(* PLC project CoDeSys External Library Template, WAGO e!COCKPIT e!COCKPIT, author 3S - Smart Software Solutions GmbH *)
(* stored: creationDateTime 2019-10-29T12:37:19.6730838, version 3.5.5.30, modificationDateTime 2019-10-29T12:36:39.3744516, organization 3S - Smart Software Solutions GmbH *)
(* Library project template with all possible element types, docu and a sample project structure *)

FUNCTION_BLOCK fbPPPSFriskoATTOM1S
  VAR_INPUT
    sKomunikat : alSTRINGKomunikat;  (* komunikat z systemu zewnętrznego *)
    intTablicaKomunikatowRozmiar : INT;  (* rozmiar tablicy danych wysyłkowych *)
    intModbusOdczytZapisZadanieRozmiar : INT;  (* rozmiar tablicy danych modbusa *)
    xTablicaKomunikatowHold : BOOL;  (* wstrzymanie komunikacji mniej ważnych komunikatów *)
    sIdInstancji : STRING;  (* parametr ID rolety np NS02L*202IBM**** *)
    sIdAplikacji : STRING;  (* parametr ID aplikacji np SO*******ECL*000 *)
    sMnemonik : STRING;  (* mnemonik właściciela - BCB* *)
    sMACAdres : STRING;  (* MAC adres sterownika *)
    sDaneZapasowe : STRING;  (* 6 znaków zapasu *)
    tCzasOpoznieniaRestartu : TIME;  (* czas opóźnienia po którym zaczynają być raportowane wartości *)
    tCzasOpoznieniaAlarmu : TIME := TIME#1m0s0ms;  (* czas opóźnienia po którym zaczynają być raportowane wartości *)
    bAdres : BYTE;
    tMinimalnyCzasRaportowania : TIME;
    tMaksymalnyCzasRaportowania : TIME;
    xAutonomizacja : BOOL;
    xAutonomizacjaSztuczna : BOOL;
    xSezonGrzewczyCalyRok : BOOL;
    rTemperaturaZasilaniaZadanaObieguCOKomfortAutonomizacja : REAL;  (* Domyślna wartość nastawy temperatury obiegu c.o. w trybie komfortowym *)
    rTemperaturaZasilaniaZadanaObieguCOEkonomicznaAutonomizacja : REAL;  (* Domyślna wartość nastawy temperatury obiegu c.o. w trybie ekonomicznym *)
  END_VAR
  VAR_IN_OUT
    arModbusOdczytCykliczny : ARRAY[1..5000] OF typModbusOdczytCykliczny;
    arModbusStatusKomunikacji : ARRAY[1..256] OF INT;
    arModbusOdczytZapisZadanie : ARRAY[1..1000] OF typModbusOdczytZapisZadanie;
    intModbusOdczytZapisZadanieZnacznikZapisu : INT;
    arTablicaKomunikatow : alARRAYTablicaKomunikatow;
    intTablicaKomunikatowZnacznikZapisu : INT;
    aTemperatury : ARRAY[0..96] OF REAL;  (* Tablica pomiarów temperatur bieżącego dnia *)
    rTemperaturaSrednia1Dzien : REAL;  (* Średnia dzienna temperatura *)
    iTemperaturyIndex : INT;  (* Index tablicy *)
    aTemperaturySrednie : ARRAY[0..2] OF REAL;  (* Tablica zawierająca średnie temperatury z trzech ostatnich dni *)
    iTemperaturySrednieIndex : INT;  (* Index tablicy śrenich temperatur *)
    rTemperaturaSrednia3Dni : REAL;  (* Średnia temperatura z trzech dni *)
    xTemperaturaSrednia3DniObliczona : BOOL;  (* Prawda, jeśli obliczona została średnia temperatura z trzech dni *)
  END_VAR
  VAR
    xPoInicjalizacji : BOOL := FALSE;  (* Inicjalizacja *)
    fbInicjalizacyjnyTimer : TON;
    tCzasInicjalizacji : TIME := TIME#30s0ms;
    xPierwszySkan : BOOL := TRUE;  (* Definicje zmiennych do odczytu wartości z modbusa *)
    intPetlaPierwszySkan : INT := 1;
    sDane : alSTRINGKomunikat;  (* Definicje do komunikacji z IZE *)
    sWyslanyKomunikat : alSTRINGKomunikat;
    sWyslanyKomunikatDummy : alSTRINGKomunikat;
    xZadanieRaportu : BOOL;
    sKomunikatPamiec : alSTRINGKomunikat;
    intPetla : INT;
    arErrorStan : ARRAY[0..10] OF INT;  (* tablica przechowująca statusy alarmowe *)
    arErrorKlasa : ARRAY[0..10] OF INT;  (* tablica przechowująca klasy danych alarmów *)
    xRaport : BOOL := FALSE;
    sTempWartoscAtrybutu : STRING;
    xOverFlow : BOOL;
    rtrigPrzywrocDomyslne : R_TRIG;  (* Przywracanie domyślnych wartości nastaw *)
    rtrigZapisModbus : R_TRIG;  (* Triger zapisu danych po Modbusie *)
    fbTaktowanieZapisywaniaModbus : TON;  (* Cykliczne żądanie zapisu danych do urządzenia *)
    fbTimerBrakuKomunikacji : TON;  (* Kontrola komunikacji urządzenia *)
    xBrakKomunikacjiPLC : BOOL;
    xBrakKomunikacjiIZE : BOOL;
    intBlokadaWykonywaniaRozkazow : INT;  (* Parametry *)
    intBlokadaWykonywaniaRozkazowZaraportowana : INT;
    wTemperaturaZasilaniaObieguCO : WORD;  (* Zmierzona temperatura wody instalacyjnej w obwodzie CO. *)
    rTemperaturaZasilaniaObieguCO : REAL;
    fbTemperaturaZasilaniaObieguCO : fbFiltrWartoscAnalogowa;
    rTemperaturaZasilaniaObieguCOZaraportowana : REAL;
    rTemperaturaZasilaniaObieguCOPamiec : REAL;  (* Sprawdzanie sprawności czujnika temperatury zasilania obwodu CO. *)
    xBrakZmianyTemperaturyZasilaniaObieguCO : BOOL;
    fbBrakZmianyTemperaturyZasilaniaObieguCOTimer : TON;
    xBladBrakZmianyTemperaturyZasilaniaObieguCO : BOOL;
    wTemperaturaZadanaObieguCO : WORD;  (* Wyliczona zadana temperatura wody instalacyjnej w obwodzie CO. *)
    rTemperaturaZadanaObieguCO : REAL;
    rTemperaturaZadanaObieguCOZaraportowana : REAL;
    xBrakOsiagnieciaTemperauryZadanejCO : BOOL;  (* Sprawdzanie czy została osiągnęta zadana temperatura zasilania obwodu CO. *)
    fbBrakOsiagnieciaTemperauryZadanejCOTimer : TON;
    xBladBrakOsiagnieciaTemperauryZadanejCO : BOOL;
    wTemperaturaZasilania : WORD;  (* Zmierzona temperatura zasilania w punkcie Tzas. *)
    rTemperaturaZasilania : REAL;
    fbTemperaturaZasilania : fbFiltrWartoscAnalogowa;
    rTemperaturaZasilaniaZaraportowana : REAL;
    wTemperaturaZewnetrzna : WORD;  (* Zmierzona temperatura zewnętrzna. *)
    rTemperaturaZewnetrzna : REAL;
    fbTemperaturaZewnetrzna : fbFiltrWartoscAnalogowa;
    rTemperaturaZewnetrznaZaraportowana : REAL;
    rTemperaturaZewnetrznaPamiec : REAL;  (* Sprawdzanie sprawności czujnika temperatury zewnętrznej. *)
    xBrakZmianyTemperaturyZewnetrznej : BOOL;
    fbBrakZmianyTemperaturyZewnetrznejTimer : TON;
    xBladBrakZmianyTemperaturyZewnetrznej : BOOL;
    wTemperaturaZewnetrznaSrednia : WORD;  (* Średnia krótkoterminowa temperatury zewnętrznej z ostatnich 2 godzin. *)
    rTemperaturaZewnetrznaSrednia : REAL;
    fbTemperaturaZewnetrznaSrednia : fbFiltrWartoscAnalogowa;
    rTemperaturaZewnetrznaSredniaZaraportowana : REAL;
    wProgram : WORD;  (* Aktywny program pracy regulatora. 0-Tygodni., 1-Ferie, 2-Party. *)
    wProgramZaraportowana : WORD;
    wTemperaturaWewnetrznaZadanaKomfort : WORD;  (* Zadana temperatura wewnętrzna komfortowa. *)
    rTemperaturaWewnetrznaZadanaKomfort : REAL;
    wTemperaturaWewnetrznaZadanaEkonomiczna : WORD;  (* Zadana temperatura wewnętrzna ekonomiczna. *)
    rTemperaturaWewnetrznaZadanaEkonomiczna : REAL;
    wTemperaturaZasilaniaZadanaObieguCOKomfort : WORD;  (* Zadana komfortowa temperatura wody instalacyjnej w trybie regulacji stałowartościowej. *)
    rTemperaturaZasilaniaZadanaObieguCOKomfort : REAL;
    rTemperaturaZasilaniaZadanaObieguCOKomfortZaraportowana : REAL;
    xTemperaturaZasilaniaZadanaObieguCOKomfortZapisz : BOOL;  (* Trigger zapisu wartości w pamięci urządzenia *)
    rTemperaturaZasilaniaZadanaObieguCOKomfortZapis : REAL;  (* Wartość do zapisania w pamięci urządzenia *)
    wTemperaturaZasilaniaZadanaObieguCOEkonomiczna : WORD;  (* Zadana ekonomiczna temperatura wody instalacyjnej w trybie regulacji stałowartościowej. *)
    rTemperaturaZasilaniaZadanaObieguCOEkonomiczna : REAL;
    rTemperaturaZasilaniaZadanaObieguCOEkonomicznaZaraportowana : REAL;
    xTemperaturaZasilaniaZadanaObieguCOEkonomicznaZapisz : BOOL;  (* Trigger zapisu wartości w pamięci urządzenia *)
    rTemperaturaZasilaniaZadanaObieguCOEkonomicznaZapis : REAL;  (* Wartość do zapisania w pamięci urządzenia *)
    wAktualnyDzien : WORD;  (* Bieżący dzień tygodnia. 0 - Poniedziałek, 1 - Wtorek, ... 6 - Niedziela. *)
    wCzasGodzina : WORD;  (* Bieżący czas - godziny. *)
    wCzasMinuta : WORD;  (* Bieżący czas - minuty. *)
    wTrybPracy : WORD;  (* Tryb pracy regulatora. 0 - Zima, 1 - Lato, 2 - Auto. *)
    rTrybPracy : REAL;
    wTrybPracyZaraportowana : WORD;
    rTrybPracyAutonomizacja : REAL;  (* Domyślny tryb pracy *)
    xTrybPracyZapisz : BOOL;  (* Trigger zapisu wartości w pamięci urządzenia *)
    rTrybPracyZapis : REAL;  (* Wartość do zapisania w pamięci urządzenia *)
    wTemperaturaProguZimaLato : WORD;  (* Temperatura progu Zima/Lato. *)
    rTemperaturaProguZimaLato : REAL;
    rTemperaturaProguZimaLatoZaraportowana : REAL;
    wMinimalnaTemperaturaZasilaniaObieguCO : WORD;  (* Minimalna temperatura zasilania obwodu CO. *)
    rMinimalnaTemperaturaZasilaniaObieguCO : REAL;
    rMinimalnaTemperaturaZasilaniaObieguCOZaraportowana : REAL;
    wKrzywaGrzewcza : WORD;  (* Numer krzywej grzewczej. *)
    wPzesuniecieKrzywejGrzewczej : WORD;  (* Pionowe przesunięcie krzywej grzania. *)
    wKontrolaTemperaturyZasilania : WORD;  (* Kontrola temperatury zasilania w punkcie Tzas. 0-Nie, 1-Tak. *)
    wMaksymalnaTemperaturaZasilaniaObieguCO : WORD;  (* Maksymalna temperatura wody instalacyjnej w punkcie Tco. *)
    rMaksymalnaTemperaturaZasilaniaObieguCO : REAL;
    rMaksymalnaTemperaturaZasilaniaObieguCOZaraportowana : REAL;
    wKpRegulatoraZaworu : WORD;  (* Wzmocnienie regulatora PI sterującego siłownikiem zaworu mieszającego. *)
    wTiRegulatoraZaworu : WORD;  (* Czas całkowania regulatora PI sterującego siłownikiem zaworu mieszającego wyrażony w sekundach. *)
    wTpsRegulatoraZaworu : WORD;  (* Czas przejścia siłownika zaworu mieszającego, od pełnego otwarcia do całkowitego zamknięcia wyrażony w sekundach. *)
    wStatusCO : WORD;  (* Parametr określa status obwodu CO. Parametr ma znaczenie, gdy regulator współpracuje z regulatorem MASTER sterującym źródłem ciepła. 0-Norm, 1-Prior *)
    wZdalneSterowanie : WORD;  (* Wykorzystanie zadajnika z czujnika temperatury wewnętrznej. 0 - Komfort, 1 - Ekonomiczny, 2 - Komfort + Ekonomiczny. *)
    wTypRegulacji : WORD;  (* Typ regulacji temperatury wody instalacyjnej. 0 - Pogodowa, 1 - Stałowartościowa. *)
    wTypRegulacjiZaraportowana : WORD;
    wPompaCO : WORD;  (* Stan wyjścia sterującego pompą obiegową CO. *)
    rPompaCO : REAL;
    wPompaCOZaraportowana : WORD;
    wZaworCOZamkniecie : WORD;  (* Stan wyjść sterujących siłownikiem zaworu mieszającego CO. *)
    rZaworCOZamkniecie : REAL;
    wZaworCOZamkniecieZaraportowana : WORD;
    wZaworCOOtwarcie : WORD;  (* Stan wyjść sterujących siłownikiem zaworu mieszającego CO. *)
    rZaworCOOtwarcie : REAL;
    wZaworCOOtwarcieZaraportowana : WORD;
    fbWschodZachod : FbCalculateSunriseSunset;  (* Obliczanie wschodu i zachodu słońca *)
    fbZegar15M : TON;  (* Timer taktujący zapisywanie temperatury *)
    xObliczSrednia3Dni : BOOL;  (* Triger obliczania średniej dziennej temperatury z 3 ostatnich dni *)
    iIloscPomiarow : INT;  (* Ilość pomiarów dokonanych w ciągu dnia *)
    rTemperaturaSrednia1DzienZaraportowana : REAL;  (* Średnia dzienna temperatura zaraporotawana *)
    xSezonGrzewczy : BOOL;  (* Włączenie ogrzewania *)
    xSezonGrzewczyZaraportowana : BOOL;  (* Włączenie ogrzewania zaraportowane *)
    xBladIloscPomiarowTemperatury : BOOL;  (* Zbyt mała ilość pomiarów dokonanych w ciągu dnia do obliczenia średniej *)
  END_VAR

            (*			
Autor:					Jan Bartczak, 2019-01-08 
Prawa majątkowe: 		Solwena Sp. z o.o., 
Aktualizacje:			2019-01-25-AWy: usunięcie buga: błędny odczyt wTemperaturaZadanaObieguCO
						2019-01-31-AWy: powiększenie liczby odzcytywanych rejestrów, wysyłanie atrybutów do IZE, konwersja danych dla dataloggera
						2019-02-05-AWy: kontrola komunikacji
						2019-02-18-AWy: generowanie alarmów od czujnika temp. zew., zasilania CO oraz braku osiągnięcia temperatury zadanej.
						2019-04-15-AWy: obsługa trybu pracy (zima/lato) z IZE
						2019-04-18-AWy: - usunięcie buga z warunku na wysłanie ramki z deaktywacją alarmu o braku osiągnięcia temperatury zadanej. 
										- dopisanie warunku pracy węzła w trybie ZIMA lub AUTO na gerenowanie w/w alarmu 
						2019-05-14-AWy: - zmiana obsługi ramki C z nastawą temperatury komfortowej i ekonomicznej.
										- zmiana adresu rejestrów temperatury zadanej CO komfort i ekonomicznej oraz tempearatury wewnętrznej komfort i ekonomicznej.
						2019-05-16-AWy: modyfikacja warunku na raportowanie. Dopisane: AND arModbusStatusKomunikacji[bAdres] = enumModbusStatus.KomunikacjaPrawidlowa AND xPoInicjalizacji 
						2019-05-17-AWy: usunięcie mnożenia *10 atrybutów TEMPNASCOKMF i TEMPNASCOEKO po otrzymaniu ramki C z tymi atrybutami.
						2019-05-22-AWy: zapisywanie po MODBUSie trybu pracy na urządzenie.
						2019-06-04-AWy: załadowanie domyślnych trybów pracy i nastaw po przejściu w tryb autonomizacji.
						2019-08-05-AWy: wyznaczanie okresu grzewczego. Wysyłanie xSezonGrzewczy i rTemperaturaSrednia1Dzien do IZE. Przeniesie xTrybPracyAutonomizacja z VAR_INPUT do VAR.
						2019-09-16-AWy: wysyłanie ramki z trybem pracy.
						2019-10-11-AWy: wprowadzenie zabezpieczenia przed przekroczeniem rozmiaru tablicy w przypadku utrary zasilania przez sterownik na całą noc.
						2019-10-22-AWy: - wydłużenie czasu fbTaktowanieZapisywaniaModbus oraz wprowadzenie trigera zapisu po Modbusie
										- zmiana trigera fbTimerBrakuKomunikacji
						
Opis:					fb służy do komunikacji z sterownikami węzłów FRISKO ATTO-M1
						W tej chwili możliwość sterowania (zapisu) rejestrów wTemperaturaZasilaniaZadanaObieguCOKomfort i wTemperaturaZasilaniaZadanaObieguCOEkonomiczna. Pozostałe tylko do odczytu.
				
*)

// Inicjalizacja sterownika
fbInicjalizacyjnyTimer(IN := (NOT xPoInicjalizacji AND arModbusStatusKomunikacji[bAdres] = enumModbusStatus.KomunikacjaPrawidlowa) , PT := tCzasOpoznieniaRestartu);
IF fbInicjalizacyjnyTimer.Q THEN
	rTemperaturaZasilaniaObieguCOZaraportowana := rTemperaturaZasilaniaObieguCO;
	rTemperaturaZadanaObieguCOZaraportowana := rTemperaturaZadanaObieguCO;
	rTemperaturaZasilaniaZaraportowana := rTemperaturaZasilania;
	rTemperalaniaZadanaObieguCOEkonomiczna;
	rTemperaturaProguZimaLatoZaraportowana := rTemperaturaProguZimaLato;
	rMinimalnaTemperaturaZasilaniaObieguCOZaraportowana := rMinimalnaTemperaturaZasilaniaObieguCO;
	rMaksymalnaTemperaturaZasilaniaObieguCOZaraportowana := rMaksymalnaTemperaturaZasilaniaObieguCO;
	wTypRegulacjiZaraportowana := wTypRegulacji;
	wPompaCOZaraportowana := wPompaCO;
	wZaworCOZamkniecieZaraportowana := wZaworCOZamkniecie;
	wZaworCOOtwarcieZaraportowana := wZaworCOOtwarcie;
	wTrybPracyZaraportowana := wTrybPracy;
	xSezonGrzewczyZaraportowana := xSezonGrzewczy;
	rTemperaturaSrednia1DzienZaraportowana := rTemperaturaSrednia1Dzien;
	xPoInicjalizacji := TRUE;
END_IF

// Włącz autonomizację jeśli sterownik jest w stanie inicjalizacji lub nastąpiło wymuszenie autonomizacji
IF NOT xPoInicjalizacji OR xAutonomizacjaSztuczna = TRUE THEN
	xAutonomizacja := TRUE;
END_IF 

// Kontrola komunikacji
fbTimerBrakuKomunikacji(IN := arModbusStatusKomunikacji[bAdres] <> enumModbusStatus.KomunikacjaPrawidlowa, PT := T#60S);
IF fbTimerBrakuKomunikacji.Q THEN
	xBrakKomunikacjiPLC := TRUE;
ELSE
	xBrakKomunikacjiPLC := FALSE;
END_IF

IF xAutonomizacja THEN
	xBrakKoxxdf
END_IF

// Deklaracja rejestrów Modbusa
IF xPierwszySkan THEN
	xPierwszySkan := FALSE;
	WHILE arModbusOdczytCykliczny[intPetlaPierwszySkan].bAdresUrzadzenia <> 0 DO
		intPetlaPierwszySkan := intPetlaPierwszySkan + 1;
	END_WHILE

	arModbusOdczytCykliczny[intPetlaPierwszySkan].bAdresUrzadzenia := bAdres;
	arModbusOdczytCykliczny[intPetlaPierwszySkan].bFunkcja := TO_BYTE(enumModbusKodyFunkcji.OdczytNRejestrow);
	arModbudfgsdfntPetlaPierwszySkan].ltCzestotliwosc := TIME_TO_LTIME(tMinimalnyCzasRaportowania);
	arModbusOdczytCykliczny[intPetlaPierwszySkan].pZmiennaReferencyjna := ADR(wCzasMinuta);
	intPetlaPierwszySkan := intPetlaPierwszySkan + 1;	
	
	arModbusOdczytCyklifdgdfgy[intPetlaPierwszySkan].uiAdresRejestru := 4003;
	arModbusOdczytCykliczny[intPetlaPierwszySkan].ltCzestotliwosc := TIME_TO_LTIME(tMinimalnyCzasRaportowania);
	arModbusOdczytCykliczny[intPetlaPierwszySkan].pZmiennaReferencyjna := ADR(wCzasGodzina);
	intPetlaPierwszySkan := intPetlaPierwszySkan + 1;	
	
	arModbusOdczytCykliczny[intPetlaPierwszySkan].bAdresUrzadzenia := bAdres;
	arModbusOdczytCykliczny[intPetlaPierwszySkan].bFunkcja := TO_BYTE(enumModbusKodyFunkcji.OdczytNRejestrow);
	arModfPetlaPierwszySkan].pZmiennaReferencyjna := ADR(wAktualnyDzien);
	intPetlaPierwszySkan := intPetlaPierwszySkan + 1;		

	arModbusOdczytCykliczny[intPetlaPierwszySkan].bAdresUrzadzenia := bAdres;
	arModbusOdczytCykliczny[intPetlaPierwszySkan].bFunkcja := TO_BYTE(enumModbusKodyFunkcji.OdczytNRejestrow);
	arModbusOdczytCykliczny[intPetlaPierwszySkan].uiAdresRejestru := 4205;
	arModbusOdczytCykliczny[intPetlaPierwszySkan].ltCzestotliwosc := TIME_TO_LTIME(tMinimalnyCzasRaportowania);
	arModbusOdczytCykliczny[intsdfYTE(enumModbusKodyFunkcji.OdczytNRejestrow);
	arModbusOdczytCykliczny[intPetlaPierwszySkan].uiAdresRejestru := 4206;
	arModbusOdczytCykliczny[intPetlaPierwszySkan].ltCzestotliwosc := TIME_TO_LTIME(tMinimalnyCzasRaportowania);
	arModbusOdczytCykliczny[intPetlaPierwszySkan].pZmiennaReferencyjna := ADR(wTemperaturaZasilaniaZadanaObieguCOEkonomiczna);
	intPetlaPierwszySkan := ffff + 1;
	
	arModbusOdczytCykliczny[intPetlaPierwszySkan].bAdresUrzadzenia := bAdres;
	arModbusOdczytCykliczny[intPetlaPierwszySkan].bFunkcja := TO_BYTE(enumModbusKodyFunkcji.OdczytNRejestrow);
	arModbusOdczytCykliczny[intPetlaPierwszySkan].uiAdresRejestru := 4032;
	arModbusOdczytCykliczny[intPetlaPierwszySkan].ltCzestotliwosc := TIME_TO_LTIME(tMinimalnyCzasRaportowania);
	arModbusOdczytCykliczny[intPetlaPierwszySkan].pZmiennaReferencyjna := ADR(wTemperaturaZasilaniaObieguCO);
	intPetlaPierwszySkan := intPetlaPierwszySkan + 1;	
	
	arModbusOdczytCykliczny[intPetlaPierwszySkan].bAdresUrzadzenia := bAdres;
	arModbusOdczytCykliczny[intPetlaPierwszySkan].bFunkcja := TO_BYTE(enumModbusKodyFunkcji.OdczytNRejestrow);
	arModbusOdczytCykliczny[intPetlaPierwszySkan].uiAdresRejestru := 4034;
	arModbusOdczytCykliczny[intPetlaPierwszySkan].ltCzestotliwosc := TIME_TO_LTIME(tMinimalnyCzasRaportowania);
	arModbusOdczytCykliczny[intPetlaPierwszySkan].pZmiennaReferencyjna := ADR(wTemperaturaZewnetrzna);
	intPetlaPierwszySkan := intPetlaPierwszySkan + 1;	
	
	arModbusOdczytCykliczny[intPetlaPierwszySkan].bAdresUrzadzenia := bAdres;
	arModbusOdczytCykliczny[intPetlaPierwszySkan].bFunkcja := TO_BYTE(enumModbusKodyFunkcji.OdczytNRejestrow);
	arModbusOdczytCykliczny[intPetlaPierwszySkan].uiAdresRejestru := 4035;
	arModbusOdczytCykliczny[intPetlaPierwszySkan].ltCzestotliwosc := TIME_TO_LTIME(tMinimalnyCzasRaportowania);
	arModbusOdczytCykliczny[intPetlaPierwszySkan].pZmiennaReferencyjna := ADR(wTemperaturaZasilania);
	intPetlaPierwszySkan := intPetlaPierwszySkan + 1;	

	arModbusOdczytCykliczny[intPetlaPierwszySkan].bAdresUrzadzenia := bAdres;
	arModbusOdczytCykliczny[intPetlaPierwszySkan].bFunkcja := TO_BYTE(enumModbusKodyFunkcji.OdczytNRejestrow);
	arModbusOdczytCykliczny[intPetlaPierwszySkan].uiAdresRejestru := 4047;
	arModbusOdczytCykliczny[intPetlaPierwszySkan].ltCzestotliwosc := TIME_TO_LTIME(tMinimalnyCzasRaportowania);
	arModbusOdczytCykliczny[intPetlaPierwszySkan].pZmiennaReferencyjna := ADR(wPompaCO);
	intPetlaPierwszySkan := intPetlaPierwszySkan + 1;
	
	arModbusOdczytCykliczny[intPetlaPierwszySkan].bAdresUrzadzenia := bAdres;
	arModbusOdczytCykliczny[intPetlaPierwszySkan].bFunkcja := TO_BYTE(enumModbusKodyFunkcji.OdczytNRejestrow);
	arModbusOdczytCykliczny[intPetlaPierwszySkan].uiAdresRejestru := 4048;
	arModbusOdczytCykliczny[intPetlaPierwszySkan].ltCzestotliwosc := TIME_TO_LTIME(tMinimalnyCzasRaportowania);
	arModbusOdczytCykliczny[intPetlaPierwszySkan].pZmiennaReferencyjna := ADR(wZaworCOZamkniecie);
	intPetlaPierwszySkan := intPetlaPierwszySkan + 1;
	
	arModbusOdczytCykliczny[intPetlaPierwszySkan].bAdresUrzadzenia := bAdres;
	arModbusOdczytCykliczny[intPetlaPierwszySkan].bFunkcja := TO_BYTE(enumModbusKodyFunkcji.OdczytNRejestrow);
	arModbusOdczytCykliczny[intPetlaPierwszySkan].uiAdresRejestru := 4049;
	arModbusOdczytCykliczny[intPetlaPierwszySkan].ltCzestotliwosc := TIME_TO_LTIME(tMinimalnyCzasRaportowania);
	arModbusOdczytCykliczny[intPetlaPierwszySkan].pZmiennaReferencyjna := ADR(wZaworCOOtwarcie);
	intPetlaPierwszySkan := intPetlaPierwszySkan + 1;	
	
	arModbusOdczytCykliczny[intPetlaPierwszySkan].bAdresUrzadzenia := bAdres;
	arModbusOdczytCykliczny[intPetlaPierwszySkan].bFunkcja := TO_BYTE(enumModbusKodyFunkcji.OdczytNRejestrow);
	arModbusOdczytCykliczny[intPetlaPierwszySkan].uiAdresRejestru := 4088;
	arModbusOdczytCykliczny[intPetlaPierwszySkan].ltCzestotliwosc := TIME_TO_LTIME(tMinimalnyCzasRaportowania);
	arModbusOdczytCykliczny[intPetlaPierwszySkan].pZmiennaReferencyjna := ADR(wTemperaturaZadanaObieguCO);
	intPetlaPierwszySkan := intPetlaPierwszySkan + 1;	
		
	arModbusOdczytCykliczny[intPetlaPierwszySkan].bAdresUrzadzenia := bAdres;
	arModbusOdczytCykliczny[intPetlaPierwszySkan].bFunkcja := TO_BYTE(enumModbusKodyFunkcji.OdczytNRejestrow);
	arModbusOdczytCykliczny[intPetlaPierwszySkan].uiAdresRejestru := 4092;
	arModbusOdczytCykliczny[intPetlaPierwszySkan].ltCzestotliwosc := TIME_TO_LTIME(tMinimalnyCzasRaportowania);
	arModbusOdczytCykliczny[intPetlaPierwszySkan].pZmiennaReferencyjna := ADR(wTemperaturaZewnetrznaSrednia);
	intPetlaPierwszySkan := intPetlaPierwszySkan + 1;	
	
	arModbusOdczytCykliczny[intPetlaPierwszySkan].bAdresUrzadzenia := bAdres;
	arModbusOdczytCykliczny[intPetlaPierwszySkan].bFunkcja := TO_BYTE(enumModbusKodyFunkcji.OdczytNRejestrow);
	arModbusOdczytCykliczny[intPetlaPierwszySkan].uiAdresRejestru := 4124;
	arModbusOdczytCykliczny[intPetlaPierwszySkan].ltCzestotliwosc := TIME_TO_LTIME(tMinimalnyCzasRaportowania);
	arModbusOdczytCykliczny[intPetlaPierwszySkan].pZmiennaReferencyjna := ADR(wTemperaturaWewnetrznaZadanaKomfort);
	intPetlaPierwszySkan := intPetlaPierwszySkan + 1;	
		
	arModbusOdczytCykliczny[intPetlaPierwszySkan].bAdresUrzadzenia := bAdres;
	arModbusOdczytCykliczny[intPetlaPierwszySkan].bFunkcja := TO_BYTE(enumModbusKodyFunkcji.OdczytNRejestrow);
	arModbusOdczytCykliczny[intPetlaPierwszySkan].uiAdresRejestru := 4125;
	arModbusOdczytCykliczny[intPetlaPierwszySkan].ltCzestotliwosc := TIME_TO_LTIME(tMinimalnyCzasRaportowania);
	arModbusOdczytCykliczny[intPetlaPierwszySkan].pZmiennaReferencyjna := ADR(wTemperaturaWewnetrznaZadanaEkonomiczna);
	intPetlaPierwszySkan := intPetlaPierwszySkan + 1;	
	
	arModbusOdczytCykliczny[intPetlaPierwszySkan].bAdresUrzadzenia := bAdres;
	arModbusOdczytCykliczny[intPetlaPierwszySkan].bFunkcja := TO_BYTE(enumModbusKodyFunkcji.OdczytNRejestrow);
	arModbusOdczytCykliczny[intPetlaPierwszySkan].uiAdresRejestru := 4173;
	arModbusOdczytCykliczny[intPetlaPierwszySkan].ltCzestotliwosc := TIME_TO_LTIME(tMinimalnyCzasRaportowania);
	arModbusOdczytCykliczny[intPetlaPierwszySkan].pZmiennaReferencyjna := ADR(wTrybPracy);
	intPetlaPierwszySkan := intPetlaPierwszySkan + 1;	

	arModbusOdczytCykliczny[intPetlaPierwszySkan].bAdresUrzadzenia := bAdres;
	arModbusOdczytCykliczny[intPetlaPierwszySkan].bFunkcja := TO_BYTE(enumModbusKodyFunkcji.OdczytNRejestrow);
	arModbusOdczytCykliczny[intPetlaPierwszySkan].uiAdresRejestru := 4170;
	arModbusOdczytCykliczny[intPetlaPierwszySkan].ltCzestotliwosc := TIME_TO_LTIME(tMinimalnyCzasRaportowania);
	arModbusOdczytCykliczny[intPetlaPierwszySkan].pZmiennaReferencyjna := ADR(wKrzywaGrzewcza);
	intPetlaPierwszySkan := intPetlaPierwszySkan + 1;	
	
	arModbusOdczytCykliczny[intPetlaPierwszySkan].bAdresUrzadzenia := bAdres;
	arModbusOdczytCykliczny[intPetlaPierwszySkan].bFunkcja := TO_BYTE(enumModbusKodyFunkcji.OdczytNRejestrow);
	arModbusOdczytCykliczny[intPetlaPierwszySkan].uiAdresRejestru := 4174;
	arModbusOdczytCykliczny[intPetlaPierwszySkan].ltCzestotliwosc := TIME_TO_LTIME(tMinimalnyCzasRaportowania);
	arModbusOdczytCykliczny[intPetlaPierwszySkan].pZmiennaReferencyjna := ADR(wTemperaturaProguZimaLato);
	intPetlaPierwszySkan := intPetlaPierwszySkan + 1;	
	
	arModbusOdczytCykliczny[intPetlaPierwszySkan].bAdresUrzadzenia := bAdres;
	arModbusOdczytCykliczny[intPetlaPierwszySkan].bFunkcja := TO_BYTE(enumModbusKodyFunkcji.OdczytNRejestrow);
	arModbusOdczytCykliczny[intPetlaPierwszySkan].uiAdresRejestru := 4175;
	arModbusOdczytCykliczny[intPetlaPierwszySkan].ltCzestotliwosc := TIME_TO_LTIME(tMinimalnyCzasRaportowania);
	arModbusOdczytCykliczny[intPetlaPierwszySkan].pZmiennaReferencyjna := ADR(wKpRegulatoraZaworu);
	intPetlaPierwszySkan := intPetlaPierwszySkan + 1;	
			
	arModbusOdczytCykliczny[intPetlaPierwszySkan].bAdresUrzadzenia := bAdres;
	arModbusOdczytCykliczny[intPetlaPierwszySkan].bFunkcja := TO_BYTE(enumModbusKodyFunkcji.OdczytNRejestrow);
	arModbusOdczytCykliczny[intPetlaPierwszySkan].uiAdresRejestru := 4176;
	arModbusOdczytCykliczny[intPetlaPierwszySkan].ltCzestotliwosc := TIME_TO_LTIME(tMinimalnyCzasRaportowania);
	arModbusOdczytCykliczny[intPetlaPierwszySkan].pZmiennaReferencyjna := ADR(wTiRegulatoraZaworu);
	intPetlaPierwszySkan := intPetlaPierwszySkan + 1;	
	
	arModbusOdczytCykliczny[intPetlaPierwszySkan].bAdresUrzadzenia := bAdres;
	arModbusOdczytCykliczny[intPetlaPierwszySkan].bFunkcja := TO_BYTE(enumModbusKodyFunkcji.OdczytNRejestrow);
	arModbusOdczytCykliczny[intPetlaPierwszySkan].uiAdresRejestru := 4183;
	arModbusOdczytCykliczny[intPetlaPierwszySkan].ltCzestotliwosc := TIME_TO_LTIME(tMinimalnyCzasRaportowania);
	arModbusOdczytCykliczny[intPetlaPierwszySkan].pZmiennaReferencyjna := ADR(wTpsRegulatoraZaworu);
	intPetlaPierwszySkan := intPetlaPierwszySkan + 1;
	
	arModbusOdczytCykliczny[intPetlaPierwszySkan].bAdresUrzadzenia := bAdres;
	arModbusOdczytCykliczny[intPetlaPierwszySkan].bFunkcja := TO_BYTE(enumModbusKodyFunkcji.OdczytNRejestrow);
	arModbusOdczytCykliczny[intPetlaPierwszySkan].uiAdresRejestru := 4188;
	arModbusOdczytCykliczny[intPetlaPierwszySkan].ltCzestotliwosc := TIME_TO_LTIME(tMinimalnyCzasRaportowania);
	arModbusOdczytCykliczny[intPetlaPierwszySkan].pZmiennaReferencyjna := ADR(wMinimalnaTemperaturaZasilaniaObieguCO);
	intPetlaPierwszySkan := intPetlaPierwszySkan + 1;	
				
	arModbusOdczytCykliczny[intPetlaPierwszySkan].bAdresUrzadzenia := bAdres;
	arModbusOdczytCykliczny[intPetlaPierwszySkan].bFunkcja := TO_BYTE(enumModbusKodyFunkcji.OdczytNRejestrow);
	arModbusOdczytCykliczny[intPetlaPierwszySkan].uiAdresRejestru := 4189;
	arModbusOdczytCykliczny[intPetlaPierwszySkan].ltCzestotliwosc := TIME_TO_LTIME(tMinimalnyCzasRaportowania);
	arModbusOdczytCykliczny[intPetlaPierwszySkan].pZmiennaReferencyjna := ADR(wMaksymalnaTemperaturaZasilaniaObieguCO);
	intPetlaPierwszySkan := intPetlaPierwszySkan + 1;	
		
	arModbusOdczytCykliczny[intPetlaPierwszySkan].bAdresUrzadzenia := bAdres;
	arModbusOdczytCykliczny[intPetlaPierwszySkan].bFunkcja := TO_BYTE(enumModbusKodyFunkcji.OdczytNRejestrow);
	arModbusOdczytCykliczny[intPetlaPierwszySkan].uiAdresRejestru := 4191;
	arModbusOdczytCykliczny[intPetlaPierwszySkan].ltCzestotliwosc := TIME_TO_LTIME(tMinimalnyCzasRaportowania);
	arModbusOdczytCykliczny[intPetlaPierwszySkan].pZmiennaReferencyjna := ADR(wKontrolaTemperaturyZasilania);
	intPetlaPierwszySkan := intPetlaPierwszySkan + 1;	
		
	arModbusOdczytCykliczny[intPetlaPierwszySkan].bAdresUrzadzenia := bAdres;
	arModbusOdczytCykliczny[intPetlaPierwszySkan].bFunkcja := TO_BYTE(enumModbusKodyFunkcji.OdczytNRejestrow);
	arModbusOdczytCykliczny[intPetlaPierwszySkan].uiAdresRejestru := 4194;
	arModbusOdczytCykliczny[intPetlaPierwszySkan].ltCzestotliwosc := TIME_TO_LTIME(tMinimalnyCzasRaportowania);
	arModbusOdczytCykliczny[intPetlaPierwszySkan].pZmiennaReferencyjna := ADR(wPzesuniecieKrzywejGrzewczej);
	intPetlaPierwszySkan := intPetlaPierwszySkan + 1;	
	
	arModbusOdczytCykliczny[intPetlaPierwszySkan].bAdresUrzadzenia := bAdres;
	arModbusOdczytCykliczny[intPetlaPierwszySkan].bFunkcja := TO_BYTE(enumModbusKodyFunkcji.OdczytNRejestrow);
	arModbusOdczytCykliczny[intPetlaPierwszySkan].uiAdresRejestru := 4197;
	arModbusOdczytCykliczny[intPetlaPierwszySkan].ltCzestotliwosc := TIME_TO_LTIME(tMinimalnyCzasRaportowania);
	arModbusOdczytCykliczny[intPetlaPierwszySkan].pZmiennaReferencyjna := ADR(wProgram);
	intPetlaPierwszySkan := intPetlaPierwszySkan + 1;	

	arModbusOdczytCykliczny[intPetlaPierwszySkan].bAdresUrzadzenia := bAdres;
	arModbusOdczytCykliczny[intPetlaPierwszySkan].bFunkcja := TO_BYTE(enumModbusKodyFunkcji.OdczytNRejestrow);
	arModbusOdczytCykliczny[intPetlaPierwszySkan].uiAdresRejestru := 4201;
	arModbusOdczytCykliczny[intPetlaPierwszySkan].ltCzestotliwosc := TIME_TO_LTIME(tMinimalnyCzasRaportowania);
	arModbusOdczytCykliczny[intPetlaPierwszySkan].pZmiennaReferencyjna := ADR(wZdalneSterowanie);
	intPetlaPierwszySkan := intPetlaPierwszySkan + 1;
		
	arModbusOdczytCykliczny[intPetlaPierwszySkan].bAdresUrzadzenia := bAdres;
	arModbusOdczytCykliczny[intPetlaPierwszySkan].bFunkcja := TO_BYTE(enumModbusKodyFunkcji.OdczytNRejestrow);
	arModbusOdczytCykliczny[intPetlaPierwszySkan].uiAdresRejestru := 4202;
	arModbusOdczytCykliczny[intPetlaPierwszySkan].ltCzestotliwosc := TIME_TO_LTIME(tMinimalnyCzasRaportowania);
	arModbusOdczytCykliczny[intPetlaPierwszySkan].pZmiennaReferencyjna := ADR(wStatusCO);
	intPetlaPierwszySkan := intPetlaPierwszySkan + 1;			
	
	arModbusOdczytCykliczny[intPetlaPierwszySkan].bAdresUrzadzenia := bAdres;
	arModbusOdczytCykliczny[intPetlaPierwszySkan].bFunkcja := TO_BYTE(enumModbusKodyFunkcji.OdczytNRejestrow);
	arModbusOdczytCykliczny[intPetlaPierwszySkan].uiAdresRejestru := 4204;
	arModbusOdczytCykliczny[intPetlaPierwszySkan].ltCzestotliwosc := TIME_TO_LTIME(tMinimalnyCzasRaportowania);
	arModbusOdczytCykliczny[intPetlaPierwszySkan].pZmiennaReferencyjna := ADR(wTypRegulacji);
	intPetlaPierwszySkan := intPetlaPierwszySkan + 1;	
END_IF

// Przeliczenie zmiennych
fbTemperaturaZasilaniaObieguCO(	rWartoscWejsciowa := WORD_TO_REAL(wTemperaturaZasilaniaObieguCO),
								rDeadband := 0.5,
								tCzasMinimalny := tMinimalnyCzasRaportowania,
								tCzasMaksymalny := tMaksymalnyCzasRaportowania,
								rWynikMnoznik := 0.1,
								rWynikOffset := 273.15,
								rWartoscWejsciowaZaraportowana := rTemperaturaZasilaniaObieguCOZaraportowana,
								rWartoscWyjsciowa => rTemperaturaZasilaniaObieguCO);
								
rTemperaturaZadanaObieguCO := WORD_TO_REAL(wTemperaturaZadanaObieguCO)*0.1 + 273.15;
fbTemperaturaZasilania( rWartoscWejsciowa := WORD_TO_REAL(wTemperaturaZasilania),
						rDeadband := 0.5,
						tCzasMinimalny := tMinimalnyCzasRaportowania,
						tCzasMaksymalny := tMaksymalnyCzasRaportowania,
						rWynikMnoznik := 0.1,
						rWynikOffset := 273.15,
						rWartoscWejsciowaZaraportowana := rTemperaturaZasilaniaZaraportowana,
						rWartoscWyjsciowa => rTemperaturaZasilania);

			
fbTemperaturaZewnetrzna(	rWartoscWejsciowa := WORD_TO_REAL(wTemperaturaZewnetrzna),
							rDeadband := 0.5,
							tCzasMinimalny := tMinimalnyCzasRaportowania,
							tCzasMaksymalny := tMaksymalnyCzasRaportowania,
							rWynikMnoznik := 0.1,
							rWynikOffset := 273.15,
							rWartoscWejsciowaZaraportowana := rTemperaturaZewnetrznaZaraportowana,
							rWartoscWyjsciowa => rTemperaturaZewnetrzna);


fbTemperaturaZewnetrznaSrednia(	rWartoscWejsciowa := WORD_TO_REAL(wTemperaturaZewnetrznaSrednia),
								rDeadband := 0.5,
								tCzasMinimalny := tMinimalnyCzasRaportowania,
								tCzasMaksymalny := tMaksymalnyCzasRaportowania,
								rWynikMnoznik := 0.1,
								rWynikOffset := 273.15,
								rWartoscWejsciowaZaraportowana := rTemperaturaZewnetrznaSredniaZaraportowana,
								rWartoscWyjsciowa => rTemperaturaZewnetrznaSrednia);

rTemperaturaWewnetrznaZadanaKomfort := WORD_TO_REAL(wTemperaturaWewnetrznaZadanaKomfort) + 273.15;
rTemperaturaWewnetrznaZadanaEkonomiczna := WORD_TO_REAL(wTemperaturaWewnetrznaZadanaEkonomiczna) + 273.15;
rTemperaturaZasilaniaZadanaObieguCOKomfort := WORD_TO_REAL(wTemperaturaZasilaniaZadanaObieguCOKomfort) + 273.15;
rTemperaturaZasilaniaZadanaObieguCOEkonomiczna := WORD_TO_REAL(wTemperaturaZasilaniaZadanaObieguCOEkonomiczna) + 273.15;
rTemperaturaProguZimaLato := WORD_TO_REAL(wTemperaturaProguZimaLato) + 273.15;
rMinimalnaTemperaturaZasilaniaObieguCO := WORD_TO_REAL(wMinimalnaTemperaturaZasilaniaObieguCO) + 273.15;
rMaksymalnaTemperaturaZasilaniaObieguCO := WORD_TO_REAL(wMaksymalnaTemperaturaZasilaniaObieguCO) + 273.15;
rPompaCO := WORD_TO_REAL(wPompaCO);
rZaworCOZamkniecie := WORD_TO_REAL(wZaworCOZamkniecie);
rZaworCOOtwarcie := WORD_TO_REAL(wZaworCOOtwarcie);
rTrybPracy := WORD_TO_REAL(wTrybPracy);

// Sprawdzanie czy pomiar temperatury zewnętrznej działa (alarm jest generowany, jeśli odczyt nie zmienił wartości w przeciągu 12h)
IF rTemperaturaZewnetrznaPamiec = rTemperaturaZewnetrzna THEN
	xBrakZmianyTemperaturyZewnetrznej := TRUE;
ELSE
	xBrakZmianyTemperaturyZewnetrznej := FALSE;	
END_IF
fbBrakZmianyTemperaturyZewnetrznejTimer(IN := xBrakZmianyTemperaturyZewnetrznej, PT := T#12H);
rTemperaturaZewnetrznaPamiec := rTemperaturaZewnetrzna;
IF fbBrakZmianyTemperaturyZewnetrznejTimer.Q THEN
	xBladBrakZmianyTemperaturyZewnetrznej := TRUE;
ELSE
	xBladBrakZmianyTemperaturyZewnetrznej := FALSE;
END_IF

// Sprawdzanie czy pomiar temperatury zasilania Obiegu CO działa (alarm jest generowany, jeśli odczyt nie zmienił wartości w przeciągu 12h)
IF rTemperaturaZasilaniaObieguCOPamiec = rTemperaturaZasilaniaObieguCO THEN
	xBrakZmianyTemperaturyZasilaniaObieguCO := TRUE;
ELSE
	xBrakZmianyTemperaturyZasilaniaObieguCO := FALSE;	
END_IF
fbBrakZmianyTemperaturyZasilaniaObieguCOTimer(IN := xBrakZmianyTemperaturyZasilaniaObieguCO, PT := T#12H);
rTemperaturaZasilaniaObieguCOPamiec := rTemperaturaZasilaniaObieguCO;
IF fbBrakZmianyTemperaturyZasilaniaObieguCOTimer.Q THEN
	xBladBrakZmianyTemperaturyZasilaniaObieguCO := TRUE;
ELSE
	xBladBrakZmianyTemperaturyZasilaniaObieguCO := FALSE;
END_IF

// Sprawdzanie czy została osiągnęta zadana temperatura zasilania Obiegu CO
IF rTemperaturaZasilaniaObieguCO < rTemperaturaZadanaObieguCO AND wTrybPracy <> enumPPPSFriskoATTOM1STrybPracy.Lato THEN
	xBrakOsiagnieciaTemperauryZadanejCO := TRUE;
ELSE
	xBrakOsiagnieciaTemperauryZadanejCO := FALSE;	
END_IF
fbBrakOsiagnieciaTemperauryZadanejCOTimer(IN := xBrakOsiagnieciaTemperauryZadanejCO, PT := T#3H);
IF fbBrakOsiagnieciaTemperauryZadanejCOTimer.Q THEN
	xBladBrakOsiagnieciaTemperauryZadanejCO := TRUE;
ELSE
	xBladBrakOsiagnieciaTemperauryZadanejCO := FALSE;
END_IF

// Obsługa komunikatu przychodzacego z IZE
IF sKomunikat <> sKomunikatPamiec AND xPoInicjalizacji THEN
	sKomunikatPamiec := sKomunikat;
	IF fnIDOdbiorcyMatch(sKomunikat , sIdInstancji) THEN
		sDane := '';
		// Rozkaz typu C
		IF fnKomunikatTyp(sKomunikat) = 'C' AND NOT xAutonomizacja THEN
			// Blokada wykonywania rozkazów
			IF fnKomunikatDaneSzukajWartosci(sKomunikat,'BLOK=') = '0' THEN
				IF intBlokadaWykonywaniaRozkazow = 1 THEN
					intBlokadaWykonywaniaRozkazow := 0;
				ELSE	
					IF sDane <> '' THEN
						sDane := CONCAT(sDane , ';');
					END_IF
					sDane := CONCAT(sDane , 'BLOK=0');
				END_IF
			END_IF
			IF fnKomunikatDaneSzukajWartosci(sKomunikat,'BLOK=') = '1' THEN
				IF intBlokadaWykonywaniaRozkazow = 0 THEN
					intBlokadaWykonywaniaRozkazow := 1;
				ELSE
					IF sDane <> '' THEN
						sDane := CONCAT(sDane , ';');
					END_IF					
					sDane := CONCAT(sDane , 'BLOK=1');
				END_IF
			END_IF
			
			IF intBlokadaWykonywaniaRozkazow = 0 THEN
				// Tryby pracy 
				fnKomunikatDaneZnajdzPorownajZapisz(sKomunikat := sKomunikat,
					sAtrybut := 'TRYB=',
					rAtrybutWartosc := rTrybPracyZapis,
					sDane := sDane,
					xAtrybutZapisz => xTrybPracyZapisz);		
				// Temperatura nastawiona w trybie komfortowym
				fnKomunikatDaneZnajdzPorownajZapisz(sKomunikat := sKomunikat,
					sAtrybut := 'TEMPNASCOKMF=',
					rAtrybutWartosc := rTemperaturaZasilaniaZadanaObieguCOKomfortZapis,
					sDane := sDane,
					xAtrybutZapisz => xTemperaturaZasilaniaZadanaObieguCOKomfortZapisz);
				// Temperatura nastawiona w trybie ekonomicznym
				fnKomunikatDaneZnajdzPorownajZapisz(sKomunikat := sKomunikat,
					sAtrybut := 'TEMPNASCOEKO=',
					rAtrybutWartosc := rTemperaturaZasilaniaZadanaObieguCOEkonomicznaZapis,
					sDane := sDane,
					xAtrybutZapisz => xTemperaturaZasilaniaZadanaObieguCOEkonomicznaZapisz);
			END_IF
		END_IF

		// Zapytanie typu Q
		IF fnKomunikatTyp(sKomunikat) = 'Q' AND arModbusStatusKomunikacji[bAdres] = enumModbusStatus.KomunikacjaPrawidlowa THEN
			IF fnKomunikatDaneSzukajWartosci(sKomunikat , 'BLOK=') = '?' OR fnKomunikatDaneSzukajWartosci(sKomunikat , 'ALL=') = '?' THEN
				fnKomunikatDaneDodaj_xOverFlow(sDane := sDane , sAtrybut := 'BLOK=' , sWartosc := INT_TO_STRING(intBlokadaWykonywaniaRozkazow) , xOverFlow := xOverFlow);	
				IF xOverFlow = TRUE THEN
					fnZapiszKomunikat(	sCalyKomunikat := '' ,
								sTypKomunikatu := 'A' ,
								sMnemonik := sMnemonik ,
								sMACAdres := sMACAdres ,
								sIDNadawcy := sIdInstancji ,
								sIDOdbiorcy := sIdAplikacji ,
								sDaneZapasowe := sDaneZapasowe ,
								sDane := sDane ,
								arTablicaKomunikatow := arTablicaKomunikatow ,
								intTablicaKomunikatowZnacznikZapisu := intTablicaKomunikatowZnacznikZapisu ,
								intTablicaKomunikatowRozmiar := intTablicaKomunikatowRozmiar ,
								sWyslanyKomunikat := sWyslanyKomunikatDummy);
					sDane := '';
				END_IF
			END_IF
			IF fnKomunikatDaneSzukajWartosci(sKomunikat , 'TRYB=') = '?' OR fnKomunikatDaneSzukajWartosci(sKomunikat , 'ALL=') = '?' THEN
				fnKomunikatDaneDodaj_xOverFlow(sDane := sDane , sAtrybut := 'TRYB=' , sWartosc := REAL_TO_STRING(rTrybPracy) , xOverFlow := xOverFlow);	
				IF xOverFlow = TRUE THEN
					fnZapiszKomunikat(	sCalyKomunikat := '' ,
								sTypKomunikatu := 'A' ,
								sMnemonik := sMnemonik ,
								sMACAdres := sMACAdres ,
								sIDNadawcy := sIdInstancji ,
								sIDOdbiorcy := sIdAplikacji ,
								sDaneZapasowe := sDaneZapasowe ,
								sDane := sDane ,
								arTablicaKomunikatow := arTablicaKomunikatow ,
								intTablicaKomunikatowZnacznikZapisu := intTablicaKomunikatowZnacznikZapisu ,
								intTablicaKomunikatowRozmiar := intTablicaKomunikatowRozmiar ,
								sWyslanyKomunikat := sWyslanyKomunikatDummy);
					sDane := '';
				END_IF
			END_IF
			IF fnKomunikatDaneSzukajWartosci(sKomunikat , 'TEMPZASCO=') = '?' OR fnKomunikatDaneSzukajWartosci(sKomunikat , 'ALL=') = '?' THEN
				fnKomunikatDaneDodaj_xOverFlow(sDane := sDane , sAtrybut := 'TEMPZASCO=' , sWartosc := REAL_TO_STRING(rTemperaturaZasilaniaObieguCO) , xOverFlow := xOverFlow);	
				IF xOverFlow = TRUE THEN
					fnZapiszKomunikat(	sCalyKomunikat := '' ,
								sTypKomunikatu := 'A' ,
								sMnemonik := sMnemonik ,
								sMACAdres := sMACAdres ,
								sIDNadawcy := sIdInstancji ,
								sIDOdbiorcy := sIdAplikacji ,
								sDaneZapasowe := sDaneZapasowe ,
								sDane := sDane ,
								arTablicaKomunikatow := arTablicaKomunikatow ,
								intTablicaKomunikatowZnacznikZapisu := intTablicaKomunikatowZnacznikZapisu ,
								intTablicaKomunikatowRozmiar := intTablicaKomunikatowRozmiar ,
								sWyslanyKomunikat := sWyslanyKomunikatDummy);
					sDane := '';
				END_IF
			END_IF
			IF fnKomunikatDaneSzukajWartosci(sKomunikat , 'TEMPZADCO=') = '?' OR fnKomunikatDaneSzukajWartosci(sKomunikat , 'ALL=') = '?' THEN
				fnKomunikatDaneDodaj_xOverFlow(sDane := sDane , sAtrybut := 'TEMPZADCO=' , sWartosc := REAL_TO_STRING(rTemperaturaZadanaObieguCO) , xOverFlow := xOverFlow);	
				IF xOverFlow = TRUE THEN
					fnZapiszKomunikat(	sCalyKomunikat := '' ,
								sTypKomunikatu := 'A' ,
								sMnemonik := sMnemonik ,
								sMACAdres := sMACAdres ,
								sIDNadawcy := sIdInstancji ,
								sIDOdbiorcy := sIdAplikacji ,
								sDaneZapasowe := sDaneZapasowe ,
								sDane := sDane ,
								arTablicaKomunikatow := arTablicaKomunikatow ,
								intTablicaKomunikatowZnacznikZapisu := intTablicaKomunikatowZnacznikZapisu ,
								intTablicaKomunikatowRozmiar := intTablicaKomunikatowRozmiar ,
								sWyslanyKomunikat := sWyslanyKomunikatDummy);
					sDane := '';
				END_IF
			END_IF
			IF fnKomunikatDaneSzukajWartosci(sKomunikat , 'TEMPZAS=') = '?' OR fnKomunikatDaneSzukajWartosci(sKomunikat , 'ALL=') = '?' THEN
				fnKomunikatDaneDodaj_xOverFlow(sDane := sDane , sAtrybut := 'TEMPZAS=' , sWartosc := REAL_TO_STRING(rTemperaturaZasilania) , xOverFlow := xOverFlow);	
				IF xOverFlow = TRUE THEN
					fnZapiszKomunikat(	sCalyKomunikat := '' ,
								sTypKomunikatu := 'A' ,
								sMnemonik := sMnemonik ,
								sMACAdres := sMACAdres ,
								sIDNadawcy := sIdInstancji ,
								sIDOdbiorcy := sIdAplikacji ,
								sDaneZapasowe := sDaneZapasowe ,
								sDane := sDane ,
								arTablicaKomunikatow := arTablicaKomunikatow ,
								intTablicaKomunikatowZnacznikZapisu := intTablicaKomunikatowZnacznikZapisu ,
								intTablicaKomunikatowRozmiar := intTablicaKomunikatowRozmiar ,
								sWyslanyKomunikat := sWyslanyKomunikatDummy);
					sDane := '';
				END_IF
			END_IF
			IF fnKomunikatDaneSzukajWartosci(sKomunikat , 'TEMPZEW=') = '?' OR fnKomunikatDaneSzukajWartosci(sKomunikat , 'ALL=') = '?' THEN
				fnKomunikatDaneDodaj_xOverFlow(sDane := sDane , sAtrybut := 'TEMPZEW=' , sWartosc := REAL_TO_STRING(rTemperaturaZewnetrzna) , xOverFlow := xOverFlow);	
				IF xOverFlow = TRUE THEN
					fnZapiszKomunikat(	sCalyKomunikat := '' ,
								sTypKomunikatu := 'A' ,
								sMnemonik := sMnemonik ,
								sMACAdres := sMACAdres ,
								sIDNadawcy := sIdInstancji ,
								sIDOdbiorcy := sIdAplikacji ,
								sDaneZapasowe := sDaneZapasowe ,
								sDane := sDane ,
								arTablicaKomunikatow := arTablicaKomunikatow ,
								intTablicaKomunikatowZnacznikZapisu := intTablicaKomunikatowZnacznikZapisu ,
								intTablicaKomunikatowRozmiar := intTablicaKomunikatowRozmiar ,
								sWyslanyKomunikat := sWyslanyKomunikatDummy);
					sDane := '';
				END_IF
			END_IF
			IF fnKomunikatDaneSzukajWartosci(sKomunikat , 'TEMPZEWSR=') = '?' OR fnKomunikatDaneSzukajWartosci(sKomunikat , 'ALL=') = '?' THEN
				fnKomunikatDaneDodaj_xOverFlow(sDane := sDane , sAtrybut := 'TEMPZEWSR=' , sWartosc := REAL_TO_STRING(rTemperaturaZewnetrznaSrednia) , xOverFlow := xOverFlow);	
				IF xOverFlow = TRUE THEN
					fnZapiszKomunikat(	sCalyKomunikat := '' ,
								sTypKomunikatu := 'A' ,
								sMnemonik := sMnemonik ,
								sMACAdres := sMACAdres ,
								sIDNadawcy := sIdInstancji ,
								sIDOdbiorcy := sIdAplikacji ,
								sDaneZapasowe := sDaneZapasowe ,
								sDane := sDane ,
								arTablicaKomunikatow := arTablicaKomunikatow ,
								intTablicaKomunikatowZnacznikZapisu := intTablicaKomunikatowZnacznikZapisu ,
								intTablicaKomunikatowRozmiar := intTablicaKomunikatowRozmiar ,
								sWyslanyKomunikat := sWyslanyKomunikatDummy);
					sDane := '';
				END_IF
			END_IF
			IF fnKomunikatDaneSzukajWartosci(sKomunikat , 'PROGRAM=') = '?' OR fnKomunikatDaneSzukajWartosci(sKomunikat , 'ALL=') = '?' THEN
				fnKomunikatDaneDodaj_xOverFlow(sDane := sDane , sAtrybut := 'PROGRAM=' , sWartosc := WORD_TO_STRING(wProgram) , xOverFlow := xOverFlow);	
				IF xOverFlow = TRUE THEN
					fnZapiszKomunikat(	sCalyKomunikat := '' ,
								sTypKomunikatu := 'A' ,
								sMnemonik := sMnemonik ,
								sMACAdres := sMACAdres ,
								sIDNadawcy := sIdInstancji ,
								sIDOdbiorcy := sIdAplikacji ,
								sDaneZapasowe := sDaneZapasowe ,
								sDane := sDane ,
								arTablicaKomunikatow := arTablicaKomunikatow ,
								intTablicaKomunikatowZnacznikZapisu := intTablicaKomunikatowZnacznikZapisu ,
								intTablicaKomunikatowRozmiar := intTablicaKomunikatowRozmiar ,
								sWyslanyKomunikat := sWyslanyKomunikatDummy);
					sDane := '';
				END_IF
			END_IF
			IF fnKomunikatDaneSzukajWartosci(sKomunikat , 'TEMPZASCOZADKMF=') = '?' OR fnKomunikatDaneSzukajWartosci(sKomunikat , 'ALL=') = '?' THEN
				fnKomunikatDaneDodaj_xOverFlow(sDane := sDane , sAtrybut := 'TEMPZASCOZADKMF=' , sWartosc := REAL_TO_STRING(rTemperaturaZasilaniaZadanaObieguCOKomfort) , xOverFlow := xOverFlow);	
				IF xOverFlow = TRUE THEN
					fnZapiszKomunikat(	sCalyKomunikat := '' ,
								sTypKomunikatu := 'A' ,
								sMnemonik := sMnemonik ,
								sMACAdres := sMACAdres ,
								sIDNadawcy := sIdInstancji ,
								sIDOdbiorcy := sIdAplikacji ,
								sDaneZapasowe := sDaneZapasowe ,
								sDane := sDane ,
								arTablicaKomunikatow := arTablicaKomunikatow ,
								intTablicaKomunikatowZnacznikZapisu := intTablicaKomunikatowZnacznikZapisu ,
								intTablicaKomunikatowRozmiar := intTablicaKomunikatowRozmiar ,
								sWyslanyKomunikat := sWyslanyKomunikatDummy);
					sDane := '';
				END_IF
			END_IF
			IF fnKomunikatDaneSzukajWartosci(sKomunikat , 'TEMPZASCOZADEKO=') = '?' OR fnKomunikatDaneSzukajWartosci(sKomunikat , 'ALL=') = '?' THEN
				fnKomunikatDaneDodaj_xOverFlow(sDane := sDane , sAtrybut := 'TEMPZASCOZADEKO=' , sWartosc := REAL_TO_STRING(rTemperaturaZasilaniaZadanaObieguCOEkonomiczna) , xOverFlow := xOverFlow);	
				IF xOverFlow = TRUE THEN
					fnZapiszKomunikat(	sCalyKomunikat := '' ,
								sTypKomunikatu := 'A' ,
								sMnemonik := sMnemonik ,
								sMACAdres := sMACAdres ,
								sIDNadawcy := sIdInstancji ,
								sIDOdbiorcy := sIdAplikacji ,
								sDaneZapasowe := sDaneZapasowe ,
								sDane := sDane ,
								arTablicaKomunikatow := arTablicaKomunikatow ,
								intTablicaKomunikatowZnacznikZapisu := intTablicaKomunikatowZnacznikZapisu ,
								intTablicaKomunikatowRozmiar := intTablicaKomunikatowRozmiar ,
								sWyslanyKomunikat := sWyslanyKomunikatDummy);
					sDane := '';
				END_IF
			END_IF
			IF fnKomunikatDaneSzukajWartosci(sKomunikat , 'TEMPZIMALATO=') = '?' OR fnKomunikatDaneSzukajWartosci(sKomunikat , 'ALL=') = '?' THEN
				fnKomunikatDaneDodaj_xOverFlow(sDane := sDane , sAtrybut := 'TEMPZIMALATO=' , sWartosc := REAL_TO_STRING(rTemperaturaProguZimaLato) , xOverFlow := xOverFlow);	
				IF xOverFlow = TRUE THEN
					fnZapiszKomunikat(	sCalyKomunikat := '' ,
								sTypKomunikatu := 'A' ,
								sMnemonik := sMnemonik ,
								sMACAdres := sMACAdres ,
								sIDNadawcy := sIdInstancji ,
								sIDOdbiorcy := sIdAplikacji ,
								sDaneZapasowe := sDaneZapasowe ,
								sDane := sDane ,
								arTablicaKomunikatow := arTablicaKomunikatow ,
								intTablicaKomunikatowZnacznikZapisu := intTablicaKomunikatowZnacznikZapisu ,
								intTablicaKomunikatowRozmiar := intTablicaKomunikatowRozmiar ,
								sWyslanyKomunikat := sWyslanyKomunikatDummy);
					sDane := '';
				END_IF
			END_IF
			IF fnKomunikatDaneSzukajWartosci(sKomunikat , 'TEMPMINZASCO=') = '?' OR fnKomunikatDaneSzukajWartosci(sKomunikat , 'ALL=') = '?' THEN
				fnKomunikatDaneDodaj_xOverFlow(sDane := sDane , sAtrybut := 'TEMPMINZASCO=' , sWartosc := REAL_TO_STRING(rMinimalnaTemperaturaZasilaniaObieguCO) , xOverFlow := xOverFlow);	
				IF xOverFlow = TRUE THEN
					fnZapiszKomunikat(	sCalyKomunikat := '' ,
								sTypKomunikatu := 'A' ,
								sMnemonik := sMnemonik ,
								sMACAdres := sMACAdres ,
								sIDNadawcy := sIdInstancji ,
								sIDOdbiorcy := sIdAplikacji ,
								sDaneZapasowe := sDaneZapasowe ,
								sDane := sDane ,
								arTablicaKomunikatow := arTablicaKomunikatow ,
								intTablicaKomunikatowZnacznikZapisu := intTablicaKomunikatowZnacznikZapisu ,
								intTablicaKomunikatowRozmiar := intTablicaKomunikatowRozmiar ,
								sWyslanyKomunikat := sWyslanyKomunikatDummy);
					sDane := '';
				END_IF
			END_IF
			IF fnKomunikatDaneSzukajWartosci(sKomunikat , 'TEMPMAXZASCO=') = '?' OR fnKomunikatDaneSzukajWartosci(sKomunikat , 'ALL=') = '?' THEN
				fnKomunikatDaneDodaj_xOverFlow(sDane := sDane , sAtrybut := 'TEMPMAXZASCO=' , sWartosc := REAL_TO_STRING(rMaksymalnaTemperaturaZasilaniaObieguCO) , xOverFlow := xOverFlow);	
				IF xOverFlow = TRUE THEN
					fnZapiszKomunikat(	sCalyKomunikat := '' ,
								sTypKomunikatu := 'A' ,
								sMnemonik := sMnemonik ,
								sMACAdres := sMACAdres ,
								sIDNadawcy := sIdInstancji ,
								sIDOdbiorcy := sIdAplikacji ,
								sDaneZapasowe := sDaneZapasowe ,
								sDane := sDane ,
								arTablicaKomunikatow := arTablicaKomunikatow ,
								intTablicaKomunikatowZnacznikZapisu := intTablicaKomunikatowZnacznikZapisu ,
								intTablicaKomunikatowRozmiar := intTablicaKomunikatowRozmiar ,
								sWyslanyKomunikat := sWyslanyKomunikatDummy);
					sDane := '';
				END_IF
			END_IF
			IF fnKomunikatDaneSzukajWartosci(sKomunikat , 'TYPREG=') = '?' OR fnKomunikatDaneSzukajWartosci(sKomunikat , 'ALL=') = '?' THEN
				fnKomunikatDaneDodaj_xOverFlow(sDane := sDane , sAtrybut := 'TYPREG=' , sWartosc := WORD_TO_STRING(wTypRegulacji) , xOverFlow := xOverFlow);	
				IF xOverFlow = TRUE THEN
					fnZapiszKomunikat(	sCalyKomunikat := '' ,
								sTypKomunikatu := 'A' ,
								sMnemonik := sMnemonik ,
								sMACAdres := sMACAdres ,
								sIDNadawcy := sIdInstancji ,
								sIDOdbiorcy := sIdAplikacji ,
								sDaneZapasowe := sDaneZapasowe ,
								sDane := sDane ,
								arTablicaKomunikatow := arTablicaKomunikatow ,
								intTablicaKomunikatowZnacznikZapisu := intTablicaKomunikatowZnacznikZapisu ,
								intTablicaKomunikatowRozmiar := intTablicaKomunikatowRozmiar ,
								sWyslanyKomunikat := sWyslanyKomunikatDummy);
					sDane := '';
				END_IF
			END_IF
			IF fnKomunikatDaneSzukajWartosci(sKomunikat , 'POMPA=') = '?' OR fnKomunikatDaneSzukajWartosci(sKomunikat , 'ALL=') = '?' THEN
				fnKomunikatDaneDodaj_xOverFlow(sDane := sDane , sAtrybut := 'POMPA=' , sWartosc := WORD_TO_STRING(wPompaCO) , xOverFlow := xOverFlow);	
				IF xOverFlow = TRUE THEN
					fnZapiszKomunikat(	sCalyKomunikat := '' ,
								sTypKomunikatu := 'A' ,
								sMnemonik := sMnemonik ,
								sMACAdres := sMACAdres ,
								sIDNadawcy := sIdInstancji ,
								sIDOdbiorcy := sIdAplikacji ,
								sDaneZapasowe := sDaneZapasowe ,
								sDane := sDane ,
								arTablicaKomunikatow := arTablicaKomunikatow ,
								intTablicaKomunikatowZnacznikZapisu := intTablicaKomunikatowZnacznikZapisu ,
								intTablicaKomunikatowRozmiar := intTablicaKomunikatowRozmiar ,
								sWyslanyKomunikat := sWyslanyKomunikatDummy);
					sDane := '';
				END_IF
			END_IF
			IF fnKomunikatDaneSzukajWartosci(sKomunikat , 'ZAWORCOZAM=') = '?' OR fnKomunikatDaneSzukajWartosci(sKomunikat , 'ALL=') = '?' THEN
				fnKomunikatDaneDodaj_xOverFlow(sDane := sDane , sAtrybut := 'ZAWORCOZAM=' , sWartosc := WORD_TO_STRING(wZaworCOZamkniecie) , xOverFlow := xOverFlow);	
				IF xOverFlow = TRUE THEN
					fnZapiszKomunikat(	sCalyKomunikat := '' ,
								sTypKomunikatu := 'A' ,
								sMnemonik := sMnemonik ,
								sMACAdres := sMACAdres ,
								sIDNadawcy := sIdInstancji ,
								sIDOdbiorcy := sIdAplikacji ,
								sDaneZapasowe := sDaneZapasowe ,
								sDane := sDane ,
								arTablicaKomunikatow := arTablicaKomunikatow ,
								intTablicaKomunikatowZnacznikZapisu := intTablicaKomunikatowZnacznikZapisu ,
								intTablicaKomunikatowRozmiar := intTablicaKomunikatowRozmiar ,
								sWyslanyKomunikat := sWyslanyKomunikatDummy);
					sDane := '';
				END_IF
			END_IF
			IF fnKomunikatDaneSzukajWartosci(sKomunikat , 'ZAWORCOOTW=') = '?' OR fnKomunikatDaneSzukajWartosci(sKomunikat , 'ALL=') = '?' THEN
				fnKomunikatDaneDodaj_xOverFlow(sDane := sDane , sAtrybut := 'ZAWORCOOTW=' , sWartosc := WORD_TO_STRING(wZaworCOOtwarcie) , xOverFlow := xOverFlow);	
				IF xOverFlow = TRUE THEN
					fnZapiszKomunikat(	sCalyKomunikat := '' ,
								sTypKomunikatu := 'A' ,
								sMnemonik := sMnemonik ,
								sMACAdres := sMACAdres ,
								sIDNadawcy := sIdInstancji ,
								sIDOdbiorcy := sIdAplikacji ,
								sDaneZapasowe := sDaneZapasowe ,
								sDane := sDane ,
								arTablicaKomunikatow := arTablicaKomunikatow ,
								intTablicaKomunikatowZnacznikZapisu := intTablicaKomunikatowZnacznikZapisu ,
								intTablicaKomunikatowRozmiar := intTablicaKomunikatowRozmiar ,
								sWyslanyKomunikat := sWyslanyKomunikatDummy);
					sDane := '';
				END_IF
			END_IF
			IF fnKomunikatDaneSzukajWartosci(sKomunikat , 'SEZONGRZ=') = '?' OR fnKomunikatDaneSzukajWartosci(sKomunikat , 'ALL=') = '?' THEN
				fnKomunikatDaneDodaj_xOverFlow(sDane := sDane , sAtrybut := 'SEZONGRZ=' , sWartosc := BOOL_TO_STRING(xSezonGrzewczy) , xOverFlow := xOverFlow);	
				IF xOverFlow = TRUE THEN
					fnZapiszKomunikat(	sCalyKomunikat := '' ,
								sTypKomunikatu := 'A' ,
								sMnemonik := sMnemonik ,
								sMACAdres := sMACAdres ,
								sIDNadawcy := sIdInstancji ,
								sIDOdbiorcy := sIdAplikacji ,
								sDaneZapasowe := sDaneZapasowe ,
								sDane := sDane ,
								arTablicaKomunikatow := arTablicaKomunikatow ,
								intTablicaKomunikatowZnacznikZapisu := intTablicaKomunikatowZnacznikZapisu ,
								intTablicaKomunikatowRozmiar := intTablicaKomunikatowRozmiar ,
								sWyslanyKomunikat := sWyslanyKomunikatDummy);
					sDane := '';
				END_IF
			END_IF
			IF fnKomunikatDaneSzukajWartosci(sKomunikat , 'TEMPSR1DZ=') = '?' OR fnKomunikatDaneSzukajWartosci(sKomunikat , 'ALL=') = '?' THEN
				fnKomunikatDaneDodaj_xOverFlow(sDane := sDane , sAtrybut := 'TEMPSR1DZ=' , sWartosc := REAL_TO_STRING(rTemperaturaSrednia1Dzien + 273.15) , xOverFlow := xOverFlow);	
				IF xOverFlow = TRUE THEN
					fnZapiszKomunikat(	sCalyKomunikat := '' ,
								sTypKomunikatu := 'A' ,
								sMnemonik := sMnemonik ,
								sMACAdres := sMACAdres ,
								sIDNadawcy := sIdInstancji ,
								sIDOdbiorcy := sIdAplikacji ,
								sDaneZapasowe := sDaneZapasowe ,
								sDane := sDane ,
								arTablicaKomunikatow := arTablicaKomunikatow ,
								intTablicaKomunikatowZnacznikZapisu := intTablicaKomunikatowZnacznikZapisu ,
								intTablicaKomunikatowRozmiar := intTablicaKomunikatowRozmiar ,
								sWyslanyKomunikat := sWyslanyKomunikatDummy);
					sDane := '';
				END_IF
			END_IF
			// Pytanie o stany alarmów
			IF fnKomunikatDaneSzukajWartosci(sKomunikat , 'ALARM=') = '?' OR fnKomunikatDaneSzukajWartosci(sKomunikat , 'ALL=') = '?' THEN
				FOR intPetla := 1 TO 10 BY 1 DO
					// Raportowanie typu E (stanów alarmów) na zapytanie typu Q
					IF arErrorStan[intPetla] <> enumAlarmWartosc.StanNieznany THEN
						fnZapiszKomunikat(	sCalyKomunikat := '' ,
											sTypKomunikatu := 'E' ,
											sMnemonik := sMnemonik ,
											sMACAdres := sMACAdres ,
											sIDNadawcy := sIdInstancji ,
											sIDOdbiorcy := sIdAplikacji ,
											sDaneZapasowe := sDaneZapasowe ,
											sDane := fnKomunikatDaneErrorRetry(xAktywny := arErrorStan[intPetla] = enumAlarmWartosc.StanAlarmowy , intKlasa := arErrorKlasa[intPetla] , intNumer := intPetla),
											arTablicaKomunikatow := arTablicaKomunikatow ,
											intTablicaKomunikatowZnacznikZapisu := intTablicaKomunikatowZnacznikZapisu ,
											intTablicaKomunikatowRozmiar := intTablicaKomunikatowRozmiar ,
											sWyslanyKomunikat := sWyslanyKomunikatDummy);
					END_IF
				END_FOR
			END_IF
		END_IF
		
		// Raportowanie typu A
		IF sDane <> '' THEN
			fnZapiszKomunikat(	sCalyKomunikat := '' ,
								sTypKomunikatu := 'A' ,
								sMnemonik := sMnemonik ,
								sMACAdres := sMACAdres ,
								sIDNadawcy := sIdInstancji .
								sIDOdbiorcy := sIdAplikacji ,
								sDaneZapasowe := sDaneZapasowe ,
								sDane := sDane ,
								arTablicaKomunikatow := arTablicaKomunikatow ,
								intTablicaKomunikatowZnacznikZapisu := intTablicaKomunikatowZnacznikZapisu ,
								intTablicaKomunikatowRozmiar := intTablicaKomunikatowRozmiar ,
								sWyslanyKomunikat := sWyslanyKomunikatDummy);
		END_IF
	END_IF
END_IF

// Przywrócenie wartości domyślnych nastaw krzywej grzewczej i trybów pracy w przypadku restartu sterownika lub przejścia w stan autonomizacji (brak komunikacji z IZE)
rtrigPrzywrocDomyslne(CLK := xAutonomizacja);
IF rtrigPrzywrocDomyslne.Q THEN	
	IF rTrybPracy <> rTrybPracyAutonomizacja THEN
		rTrybPracyZapis := rTrybPracyAutonomizacja;
		xTrybPracyZapisz := TRUE;
	END_IF
	IF rTemperaturaZasilaniaZadanaObieguCOKomfort <> rTemperaturaZasilaniaZadanaObieguCOKomfortAutonomizacja THEN
		rTemperaturaZasilaniaZadanaObieguCOKomfortZapis := rTemperaturaZasilaniaZadanaObieguCOKomfortAutonomizacja;
		xTemperaturaZasilaniaZadanaObieguCOKomfortZapisz := TRUE;
	END_IF
	IF rTemperaturaZasilaniaZadanaObieguCOEkonomiczna <> rTemperaturaZasilaniaZadanaObieguCOEkonomicznaAutonomizacja THEN
		rTemperaturaZasilaniaZadanaObieguCOEkonomicznaZapis := rTemperaturaZasilaniaZadanaObieguCOEkonomicznaAutonomizacja;
		xTemperaturaZasilaniaZadanaObieguCOEkonomicznaZapisz := TRUE;
	END_IF
END_IF	

// Trigger zapisu po Modbusie
rtrigZapisModbus (CLK := xTrybPracyZapisz OR xTemperaturaZasilaniaZadanaObieguCOKomfortZapisz OR xTemperaturaZasilaniaZadanaObieguCOEkonomicznaZapisz);

// Taktowanie zapisywania po Modbusie
fbTaktowanieZapisywaniaModbus(IN := NOT fbTaktowanieZapisywaniaModbus.Q, PT := T#180S);
				
// Zapisywanie trybu pracy do pamięci urządzenia
IF xTrybPracyZapisz AND (fbTaktowanieZapisywaniaModbus.Q OR rtrigZapisModbus.Q) THEN
	fnModbusZapisRejestru(	bAdresUrzadzenia := bAdres,
							bFunkcja := INT_TO_BYTE(enumModbusKodyFunkcji.ZapisRejestru),
							uiAdresRejestru := 4173,
							pZmiennaReferencyjna := 0,
							wWartoscDoZapisania := REAL_TO_WORD(rTrybPracyZapis),
							intModbusOdczytZapisZadanieRozmiar := intModbusOdczytZapisZadanieRozmiar,
							arModbusOdczytZapisZadanie := arModbusOdczytZapisZadanie,
							intModbusOdczytZapisZadanieZnacznikZapisu := intModbusOdczytZapisZadanieZnacznikZapisu);
	IF rTrybPracy = rTrybPracyZapis THEN					
		xTrybPracyZapisz := FALSE;
	END_IF
END_IF
// Zapisywanie temperatury zasilania obiegu c.o. w trybie komfortowym do pamięci urządzenia
IF xTemperaturaZasilaniaZadanaObieguCOKomfortZapisz AND (fbTaktowanieZapisywaniaModbus.Q OR rtrigZapisModbus.Q) THEN
	fnModbusZapisRejestru(	bAdresUrzadzenia := bAdres,
							bFunkcja := INT_TO_BYTE(enumModbusKodyFunkcji.ZapisRejestru),
							uiAdresRejestru := 4205,
							pZmiennaReferencyjna := 0,
							wWartoscDoZapisania := REAL_TO_WORD(rTemperaturaZasilaniaZadanaObieguCOKomfortZapis - 273.15),
							intModbusOdczytZapisZadanieRozmiar := intModbusOdczytZapisZadanieRozmiar,
							arModbusOdczytZapisZadanie := arModbusOdczytZapisZadanie,
							intModbusOdczytZapisZadanieZnacznikZapisu := intModbusOdczytZapisZadanieZnacznikZapisu);
	IF rTemperaturaZasilaniaZadanaObieguCOKomfort = rTemperaturaZasilaniaZadanaObieguCOKomfortZapis THEN 						
		xTemperaturaZasilaniaZadanaObieguCOKomfortZapisz := FALSE;
	END_IF
END_IF
// Zapisywanie temperatury zasilania obiegu c.o. w trybie ekonomicznym do pamięci urządzenia
IF xTemperaturaZasilaniaZadanaObieguCOEkonomicznaZapisz AND (fbTaktowanieZapisywaniaModbus.Q OR rtrigZapisModbus.Q) THEN
	fnModbusZapisRejestru(	bAdresUrzadzenia := bAdres,
							bFunkcja := INT_TO_BYTE(enumModbusKodyFunkcji.ZapisRejestru),
							uiAdresRejestru := 4206,
							pZmiennaReferencyjna := 0,
							wWartoscDoZapisania := REAL_TO_WORD(rTemperaturaZasilaniaZadanaObieguCOEkonomicznaZapis - 273.15),
							intModbusOdczytZapisZadanieRozmiar := intModbusOdczytZapisZadanieRozmiar,
							arModbusOdczytZapisZadanie := arModbusOdczytZapisZadanie,
							intModbusOdczytZapisZadanieZnacznikZapisu := intModbusOdczytZapisZadanieZnacznikZapisu);
	IF rTemperaturaZasilaniaZadanaObieguCOEkonomiczna = rTemperaturaZasilaniaZadanaObieguCOEkonomicznaZapis THEN
		xTemperaturaZasilaniaZadanaObieguCOEkonomicznaZapisz := FALSE;
	END_IF
END_IF

// Wyznaczanie okresu grzewczego
fbZegar15M(IN := NOT fbZegar15M.Q AND NOT xBladBrakZmianyTemperaturyZewnetrznej, PT := T#15M);

	// Obliczenie wschodu i zachodu słońca
fbWschodZachod(dtUTC_Time := WagoAppTime.FuGetDateAndTime(),
	rTimeZone := 0,
	xDST := FALSE,
	rLatitude := 54.441944,
	rLongitude := 18.559722);

	// Zapisywanie tempratury z 15-minutowym okresem, oraz obliczanie średniej
IF fbWschodZachod.dtUTC_Time > fbWschodZachod.dtSunrise AND fbWschodZachod.dtUTC_Time < fbWschodZachod.dtSunset THEN
	IF fbZegar15M.Q OR xPierwszySkan THEN
		aTemperatury[iTemperaturyIndex] := WORD_TO_REAL(wTemperaturaZewnetrzna) / 10;
		iTemperaturyIndex := iTemperaturyIndex + 1;
	END_IF	
	xObliczSrednia3Dni := TRUE;
ELSE 
	// Obliczanie średniej temperatury dziennej
	IF iTemperaturyIndex >= 40 THEN		// Oblicz średnią temperaturę tylko, jeśli zebranych zostało przynajmniej 40 próbek
		rTemperaturaSrednia1Dzien := 0;
		iIloscPomiarow := iTemperaturyIndex;
		FOR iTemperaturyIndex := 0 TO iIloscPomiarow BY 1 DO  
			rTemperaturaSrednia1Dzien := rTemperaturaSrednia1Dzien + aTemperatury[iTemperaturyIndex];
		END_FOR
		rTemperaturaSrednia1Dzien := rTemperaturaSrednia1Dzien / iTemperaturyIndex;
		xBladIloscPomiarowTemperatury := FALSE;
	ELSE
		rTemperaturaSrednia1Dzien := 15;
		xBladIloscPomiarowTemperatury := TRUE;
	END_IF
	// Obliczanie średniej z trzech dni
	IF xObliczSrednia3Dni THEN
		aTemperaturySrednie[iTemperaturySrednieIndex] := rTemperaturaSrednia1Dzien;
		iTemperaturySrednieIndex := iTemperaturySrednieIndex + 1;
		IF iTemperaturySrednieIndex = 3 THEN 
			iTemperaturySrednieIndex := 0;
			xTemperaturaSrednia3DniObliczona := TRUE;
		END_IF
		rTemperaturaSrednia3Dni := (aTemperaturySrednie[0] + aTemperaturySrednie[1] + aTemperaturySrednie[2]) / 3; 
		xObliczSrednia3Dni := FALSE;	
	END_IF
	iTemperaturyIndex := 0;
END_IF

IF iTemperaturyIndex >= 96 THEN	// Zabezpieczenie przed przekroczeniem rozmiaru tablicy w przypadku utrary zasilania przez sterownik na całą noc
	iTemperaturyIndex := 0;
END_IF

	// Sprawdzenie warunku na włączenie ogrzewania (pomiędzy 15 września a 15 maja i/lub średnia temperatura jest poniżej 15 stopni)
IF  ((fbWschodZachod._rDay >= 15 AND fbWschodZachod._rMonth = 9) OR (fbWschodZachod._rMonth > 9 OR fbWschodZachod._rMonth < 5) OR (fbWschodZachod._rDay <= 15 AND fbWschodZachod._rMonth = 5)) OR 
	(rTemperaturaSrednia3Dni < 15 AND xTemperaturaSrednia3DniObliczona) OR xSezonGrzewczyCalyRok THEN
	xSezonGrzewczy := TRUE;
	rTrybPracyAutonomizacja := enumPPPSFriskoATTOM1STrybPracy.Zima;
ELSE
	xSezonGrzewczy := FALSE;
	rTrybPracyAutonomizacja := enumPPPSFriskoATTOM1STrybPracy.Lato;
END_IF

// Raportowanie typu M do IZE wartosci odczytanych z Modbusa	
IF (intBlokadaWykonywaniaRozkazow <> intBlokadaWykonywaniaRozkazowZaraportowana OR rTemperaturaZasilaniaObieguCO <> rTemperaturaZasilaniaObieguCOZaraportowana OR 
	rTemperaturaZadanaObieguCO <> rTemperaturaZadanaObieguCOZaraportowana OR rTemperaturaZasilania <> rTemperaturaZasilaniaZaraportowana OR rTemperaturaZewnetrzna <> rTemperaturaZewnetrznaZaraportowana OR
	rTemperaturaZewnetrznaSrednia <> rTemperaturaZewnetrznaSredniaZaraportowana OR wProgram <> wProgramZaraportowana OR 
	rTemperaturaZasilaniaZadanaObieguCOKomfort <> rTemperaturaZasilaniaZadanaObieguCOKomfortZaraportowana OR 
	rTemperaturaZasilaniaZadanaObieguCOEkonomiczna <> rTemperaturaZasilaniaZadanaObieguCOEkonomicznaZaraportowana OR rTemperaturaProguZimaLato <> rTemperaturaProguZimaLatoZaraportowana OR
	rMinimalnaTemperaturaZasilaniaObieguCO <> rMinimalnaTemperaturaZasilaniaObieguCOZaraportowana OR rMaksymalnaTemperaturaZasilaniaObieguCO <> rMaksymalnaTemperaturaZasilaniaObieguCOZaraportowana OR
	wTypRegulacji <> wTypRegulacjiZaraportowana OR wPompaCO <> wPompaCOZaraportowana OR wZaworCOZamkniecie <> wZaworCOZamkniecieZaraportowana OR wZaworCOOtwarcie <> wZaworCOOtwarcieZaraportowana OR 
	wTrybPracy <> wTrybPracyZaraportowana OR xSezonGrzewczy <> xSezonGrzewczyZaraportowana OR rTemperaturaSrednia1Dzien <> rTemperaturaSrednia1DzienZaraportowana) AND 
	arModbusStatusKomunikacji[bAdres] = enumModbusStatus.KomunikacjaPrawidlowa AND xPoInicjalizacji THEN
	xRaport := TRUE;
END_IF

IF xRaport THEN
	sDane := '';
	xRaport := FALSE;
	IF intBlokadaWykonywaniaRozkazow <> intBlokadaWykonywaniaRozkazowZaraportowana THEN 
		intBlokadaWykonywaniaRozkazowZaraportowana := intBlokadaWykonywaniaRozkazow;
		fnKomunikatDaneDodaj_xOverFlow(sDane := sDane , sAtrybut := 'BLOK=' , sWartosc := INT_TO_STRING(intBlokadaWykonywaniaRozkazow) , xOverFlow := xOverFlow);	
		IF xOverFlow = TRUE THEN
			fnZapiszKomunikat(	sCalyKomunikat := '' ,
						sTypKomunikatu := 'M' ,
						sMnemonik := sMnemonik ,
						sMACAdres := sMACAdres ,
						sIDNadawcy := sIdInstancji ,
						sIDOdbiorcy := sIdAplikacji ,
						sDaneZapasowe := sDaneZapasowe ,
						sDane := sDane ,
						arTablicaKomunikatow := arTablicaKomunikatow ,
						intTablicaKomunikatowZnacznikZapisu := intTablicaKomunikatowZnacznikZapisu ,
						intTablicaKomunikatowRozmiar := intTablicaKomunikatowRozmiar ,
						sWyslanyKomunikat := sWyslanyKomunikatDummy);
			sDane := '';
		END_IF
	END_IF			
	// Tryb pracy
	IF wTrybPracy <> wTrybPracyZaraportowana THEN
		wTrybPracyZaraportowana := wTrybPracy;
		fnKomunikatDaneDodaj_xOverFlow(sDane := sDane , sAtrybut := 'TRYB=' , sWartosc := REAL_TO_STRING(rTrybPracy) , xOverFlow := xOverFlow);	
		IF xOverFlow = TRUE THEN
			fnZapiszKomunikat(	sCalyKomunikat := '' ,
						sTypKomunikatu := 'M' ,
						sMnemonik := sMnemonik ,
						sMACAdres := sMACAdres ,
						sIDNadawcy := sIdInstancji ,
						sIDOdbiorcy := sIdAplikacji ,
						sDaneZapasowe := sDaneZapasowe ,
						sDane := sDane ,
						arTablicaKomunikatow := arTablicaKomunikatow ,
						intTablicaKomunikatowZnacznikZapisu := intTablicaKomunikatowZnacznikZapisu ,
						intTablicaKomunikatowRozmiar := intTablicaKomunikatowRozmiar ,
						sWyslanyKomunikat := sWyslanyKomunikatDummy);
			sDane := '';
		END_IF	
	END_IF		
	// Temperatura zasilania obwodu c. o.
	IF rTemperaturaZasilaniaObieguCO <> rTemperaturaZasilaniaObieguCOZaraportowana THEN
		rTemperaturaZasilaniaObieguCOZaraportowana := rTemperaturaZasilaniaObieguCO;
		fnKomunikatDaneDodaj_xOverFlow(sDane := sDane , sAtrybut := 'TEMPZASCO=' , sWartosc := REAL_TO_STRING(rTemperaturaZasilaniaObieguCO) , xOverFlow := xOverFlow);	
		IF xOverFlow = TRUE THEN
			fnZapiszKomunikat(	sCalyKomunikat := '' ,
						sTypKomunikatu := 'M' ,
						sMnemonik := sMnemonik ,
						sMACAdres := sMACAdres ,
						sIDNadawcy := sIdInstancji ,
						sIDOdbiorcy := sIdAplikacji ,
						sDaneZapasowe := sDaneZapasowe ,
						sDane := sDane ,
						arTablicaKomunikatow := arTablicaKomunikatow ,
						intTablicaKomunikatowZnacznikZapisu := intTablicaKomunikatowZnacznikZapisu ,
						intTablicaKomunikatowRozmiar := intTablicaKomunikatowRozmiar ,
						sWyslanyKomunikat := sWyslanyKomunikatDummy);
			sDane := '';
		END_IF	
	END_IF
	// Temperatura zadana obwodu c. o.
	IF rTemperaturaZadanaObieguCO <> rTemperaturaZadanaObieguCOZaraportowana THEN
		rTemperaturaZadanaObieguCOZaraportowana := rTemperaturaZadanaObieguCO;
		fnKomunikatDaneDodaj_xOverFlow(sDane := sDane , sAtrybut := 'TEMPZADCO=' , sWartosc := REAL_TO_STRING(rTemperaturaZadanaObieguCO) , xOverFlow := xOverFlow);	
		IF xOverFlow = TRUE THEN
			fnZapiszKomunikat(	sCalyKomunikat := '' ,
						sTypKomunikatu := 'M' ,
						sMnemonik := sMnemonik ,
						sMACAdres := sMACAdres ,
						sIDNadawcy := sIdInstancji ,
						sIDOdbiorcy := sIdAplikacji ,
						sDaneZapasowe := sDaneZapasowe ,
						sDane := sDane ,
						arTablicaKomunikatow := arTablicaKomunikatow ,
						intTablicaKomunikatowZnacznikZapisu := intTablicaKomunikatowZnacznikZapisu ,
						intTablicaKomunikatowRozmiar := intTablicaKomunikatowRozmiar ,
						sWyslanyKomunikat := sWyslanyKomunikatDummy);
			sDane := '';
		END_IF	
	END_IF
	// Temperatura zasilania budynku
	IF rTemperaturaZasilania <> rTemperaturaZasilaniaZaraportowana THEN
		rTemperaturaZasilaniaZaraportowana := rTemperaturaZasilania;
		fnKomunikatDaneDodaj_xOverFlow(sDane := sDane , sAtrybut := 'TEMPZAS=' , sWartosc := REAL_TO_STRING(rTemperaturaZasilania) , xOverFlow := xOverFlow);	
		IF xOverFlow = TRUE THEN
			fnZapiszKomunikat(	sCalyKomunikat := '' ,
						sTypKomunikatu := 'M' ,
						sMnemonik := sMnemonik ,
						sMACAdres := sMACAdres ,
						sIDNadawcy := sIdInstancji ,
						sIDOdbiorcy := sIdAplikacji ,
						sDaneZapasowe := sDaneZapasowe ,
						sDane := sDane ,
						arTablicaKomunikatow := arTablicaKomunikatow ,
						intTablicaKomunikatowZnacznikZapisu := intTablicaKomunikatowZnacznikZapisu ,
						intTablicaKomunikatowRozmiar := intTablicaKomunikatowRozmiar ,
						sWyslanyKomunikat := sWyslanyKomunikatDummy);
			sDane := '';
		END_IF	
	END_IF
	// Temperatura zewnętrzna
	IF rTemperaturaZewnetrzna <> rTemperaturaZewnetrznaZaraportowana THEN
		rTemperaturaZewnetrznaZaraportowana := rTemperaturaZewnetrzna;
		fnKomunikatDaneDodaj_xOverFlow(sDane := sDane , sAtrybut := 'TEMPZEW=' , sWartosc := REAL_TO_STRING(rTemperaturaZewnetrzna) , xOverFlow := xOverFlow);	
		IF xOverFlow = TRUE THEN
			fnZapiszKomunikat(	sCalyKomunikat := '' ,
						sTypKomunikatu := 'M' ,
						sMnemonik := sMnemonik ,
						sMACAdres := sMACAdres ,
						sIDNadawcy := sIdInstancji ,
						sIDOdbiorcy := sIdAplikacji ,
						sDaneZapasowe := sDaneZapasowe ,
						sDane := sDane ,
						arTablicaKomunikatow := arTablicaKomunikatow ,
						intTablicaKomunikatowZnacznikZapisu := intTablicaKomunikatowZnacznikZapisu ,
						intTablicaKomunikatowRozmiar := intTablicaKomunikatowRozmiar ,
						sWyslanyKomunikat := sWyslanyKomunikatDummy);
			sDane := '';
		END_IF	
	END_IF
	// Temperatura zewnętrzna średnia (2 godz.)
	IF rTemperaturaZewnetrznaSrednia <> rTemperaturaZewnetrznaSredniaZaraportowana THEN
		rTemperaturaZewnetrznaSredniaZaraportowana := rTemperaturaZewnetrznaSrednia;
		fnKomunikatDaneDodaj_xOverFlow(sDane := sDane , sAtrybut := 'TEMPZEWSR=' , sWartosc := REAL_TO_STRING(rTemperaturaZewnetrznaSrednia) , xOverFlow := xOverFlow);	
		IF xOverFlow = TRUE THEN
			fnZapiszKomunikat(	sCalyKomunikat := '' ,
						sTypKomunikatu := 'M' ,
						sMnemonik := sMnemonik ,
						sMACAdres := sMACAdres ,
						sIDNadawcy := sIdInstancji ,
						sIDOdbiorcy := sIdAplikacji ,
						sDaneZapasowe := sDaneZapasowe ,
						sDane := sDane ,
						arTablicaKomunikatow := arTablicaKomunikatow ,
						intTablicaKomunikatowZnacznikZapisu := intTablicaKomunikatowZnacznikZapisu ,
						intTablicaKomunikatowRozmiar := intTablicaKomunikatowRozmiar ,
						sWyslanyKomunikat := sWyslanyKomunikatDummy);
			sDane := '';
		END_IF	
	END_IF
	// Program pracy regulatora
	IF wProgram <> wProgramZaraportowana THEN
		wProgramZaraportowana := wProgram;
		fnKomunikatDaneDodaj_xOverFlow(sDane := sDane , sAtrybut := 'PROGRAM=' , sWartosc := WORD_TO_STRING(wProgram) , xOverFlow := xOverFlow);	
		IF xOverFlow = TRUE THEN
			fnZapiszKomunikat(	sCalyKomunikat := '' ,
						sTypKomunikatu := 'M' ,
						sMnemonik := sMnemonik ,
						sMACAdres := sMACAdres ,
						sIDNadawcy := sIdInstancji ,
						sIDOdbiorcy := sIdAplikacji ,
						sDaneZapasowe := sDaneZapasowe ,
						sDane := sDane ,
						arTablicaKomunikatow := arTablicaKomunikatow ,
						intTablicaKomunikatowZnacznikZapisu := intTablicaKomunikatowZnacznikZapisu ,
						intTablicaKomunikatowRozmiar := intTablicaKomunikatowRozmiar ,
						sWyslanyKomunikat := sWyslanyKomunikatDummy);
			sDane := '';
		END_IF	
	END_IF
	// Zadana komfortowa temperatura wody instalacyjnej w trybie regulacji stałowartościowej
	IF rTemperaturaZasilaniaZadanaObieguCOKomfort <> rTemperaturaZasilaniaZadanaObieguCOKomfortZaraportowana THEN
		rTemperaturaZasilaniaZadanaObieguCOKomfortZaraportowana := rTemperaturaZasilaniaZadanaObieguCOKomfort;
		fnKomunikatDaneDodaj_xOverFlow(sDane := sDane , sAtrybut := 'TEMPNASCOKMF=' , sWartosc := REAL_TO_STRING(rTemperaturaZasilaniaZadanaObieguCOKomfort) , xOverFlow := xOverFlow);	
		IF xOverFlow = TRUE THEN
			fnZapiszKomunikat(	sCalyKomunikat := '' ,
						sTypKomunikatu := 'M' ,
						sMnemonik := sMnemonik ,
						sMACAdres := sMACAdres ,
						sIDNadawcy := sIdInstancji ,
						sIDOdbiorcy := sIdAplikacji ,
						sDaneZapasowe := sDaneZapasowe ,
						sDane := sDane ,
						arTablicaKomunikatow := arTablicaKomunikatow ,
						intTablicaKomunikatowZnacznikZapisu := intTablicaKomunikatowZnacznikZapisu ,
						intTablicaKomunikatowRozmiar := intTablicaKomunikatowRozmiar ,
						sWyslanyKomunikat := sWyslanyKomunikatDummy);
			sDane := '';
		END_IF	
	END_IF
	// Zadana ekonomiczna temperatura wody instalacyjnej w trybie regulacji stałowartościowej
	IF rTemperaturaZasilaniaZadanaObieguCOEkonomiczna <> rTemperaturaZasilaniaZadanaObieguCOEkonomicznaZaraportowana THEN
		rTemperaturaZasilaniaZadanaObieguCOEkonomicznaZaraportowana := rTemperaturaZasilaniaZadanaObieguCOEkonomiczna;
		fnKomunikatDaneDodaj_xOverFlow(sDane := sDane , sAtrybut := 'TEMPNASCOEKO=' , sWartosc := REAL_TO_STRING(rTemperaturaZasilaniaZadanaObieguCOEkonomiczna) , xOverFlow := xOverFlow);	
		IF xOverFlow = TRUE THEN
			fnZapiszKomunikat(	sCalyKomunikat := '' ,
						sTypKomunikatu := 'M' ,
						sMnemonik := sMnemonik ,
						sMACAdres := sMACAdres ,
						sIDNadawcy := sIdInstancji ,
						sIDOdbiorcy := sIdAplikacji ,
						sDaneZapasowe := sDaneZapasowe ,
						sDane := sDane ,
						arTablicaKomunikatow := arTablicaKomunikatow ,
						intTablicaKomunikatowZnacznikZapisu := intTablicaKomunikatowZnacznikZapisu ,
						intTablicaKomunikatowRozmiar := intTablicaKomunikatowRozmiar ,
						sWyslanyKomunikat := sWyslanyKomunikatDummy);
			sDane := '';
		END_IF	
	END_IF
	// Temperatura zasilania
	IF rTemperaturaProguZimaLato <> rTemperaturaProguZimaLatoZaraportowana THEN
		rTemperaturaProguZimaLatoZaraportowana := rTemperaturaProguZimaLato;
		fnKomunikatDaneDodaj_xOverFlow(sDane := sDane , sAtrybut := 'TEMPZIMALATO=' , sWartosc := REAL_TO_STRING(rTemperaturaProguZimaLato) , xOverFlow := xOverFlow);	
		IF xOverFlow = TRUE THEN
			fnZapiszKomunikat(	sCalyKomunikat := '' ,
						sTypKomunikatu := 'M' ,
						sMnemonik := sMnemonik ,
						sMACAdres := sMACAdres ,
						sIDNadawcy := sIdInstancji ,
						sIDOdbiorcy := sIdAplikacji ,
						sDaneZapasowe := sDaneZapasowe ,
						sDane := sDane ,
						arTablicaKomunikatow := arTablicaKomunikatow ,
						intTablicaKomunikatowZnacznikZapisu := intTablicaKomunikatowZnacznikZapisu ,
						intTablicaKomunikatowRozmiar := intTablicaKomunikatowRozmiar ,
						sWyslanyKomunikat := sWyslanyKomunikatDummy);
			sDane := '';
		END_IF	
	END_IF
	// Minimalna temperatura zasilania obwodu CO
	IF rMinimalnaTemperaturaZasilaniaObieguCO <> rMinimalnaTemperaturaZasilaniaObieguCOZaraportowana THEN
		rMinimalnaTemperaturaZasilaniaObieguCOZaraportowana := rMinimalnaTemperaturaZasilaniaObieguCO;
		fnKomunikatDaneDodaj_xOverFlow(sDane := sDane , sAtrybut := 'TEMPMINZASCO=' , sWartosc := REAL_TO_STRING(rMinimalnaTemperaturaZasilaniaObieguCO) , xOverFlow := xOverFlow);	
		IF xOverFlow = TRUE THEN
			fnZapiszKomunikat(	sCalyKomunikat := '' ,
						sTypKomunikatu := 'M' ,
						sMnemonik := sMnemonik ,
						sMACAdres := sMACAdres ,
						sIDNadawcy := sIdInstancji ,
						sIDOdbiorcy := sIdAplikacji ,
						sDaneZapasowe := sDaneZapasowe ,
						sDane := sDane ,
						arTablicaKomunikatow := arTablicaKomunikatow ,
						intTablicaKomunikatowZnacznikZapisu := intTablicaKomunikatowZnacznikZapisu ,
						intTablicaKomunikatowRozmiar := intTablicaKomunikatowRozmiar ,
						sWyslanyKomunikat := sWyslanyKomunikatDummy);
			sDane := '';
		END_IF	
	END_IF
	// Maksymalna temperatura wody instalacyjnej w punkcie Tco
	IF rMaksymalnaTemperaturaZasilaniaObieguCO <> rMaksymalnaTemperaturaZasilaniaObieguCOZaraportowana THEN
		rMaksymalnaTemperaturaZasilaniaObieguCOZaraportowana := rMaksymalnaTemperaturaZasilaniaObieguCO;
		fnKomunikatDaneDodaj_xOverFlow(sDane := sDane , sAtrybut := 'TEMPMAXZASCO=' , sWartosc := REAL_TO_STRING(rMaksymalnaTemperaturaZasilaniaObieguCO) , xOverFlow := xOverFlow);	
		IF xOverFlow = TRUE THEN
			fnZapiszKomunikat(	sCalyKomunikat := '' ,
						sTypKomunikatu := 'M' ,
						sMnemonik := sMnemonik ,
						sMACAdres := sMACAdres ,
						sIDNadawcy := sIdInstancji ,
						sIDOdbiorcy := sIdAplikacji ,
						sDaneZapasowe := sDaneZapasowe ,
						sDane := sDane ,
						arTablicaKomunikatow := arTablicaKomunikatow ,
						intTablicaKomunikatowZnacznikZapisu := intTablicaKomunikatowZnacznikZapisu ,
						intTablicaKomunikatowRozmiar := intTablicaKomunikatowRozmiar ,
						sWyslanyKomunikat := sWyslanyKomunikatDummy);
			sDane := '';
		END_IF	
	END_IF
	// Typ regulacji temperatury wody instalacyjnej
	IF wTypRegulacji <> wTypRegulacjiZaraportowana THEN
		wTypRegulacjiZaraportowana := wTypRegulacji;
		fnKomunikatDaneDodaj_xOverFlow(sDane := sDane , sAtrybut := 'TYPREG=' , sWartosc := WORD_TO_STRING(wTypRegulacji) , xOverFlow := xOverFlow);	
		IF xOverFlow = TRUE THEN
			fnZapiszKomunikat(	sCalyKomunikat := '' ,
						sTypKomunikatu := 'M' ,
						sMnemonik := sMnemonik ,
						sMACAdres := sMACAdres ,
						sIDNadawcy := sIdInstancji ,
						sIDOdbiorcy := sIdAplikacji ,
						sDaneZapasowe := sDaneZapasowe ,
						sDane := sDane ,
						arTablicaKomunikatow := arTablicaKomunikatow ,
						intTablicaKomunikatowZnacznikZapisu := intTablicaKomunikatowZnacznikZapisu ,
						intTablicaKomunikatowRozmiar := intTablicaKomunikatowRozmiar ,
						sWyslanyKomunikat := sWyslanyKomunikatDummy);
			sDane := '';
		END_IF	
	END_IF
	// Stan wyjścia sterującego pompą obiegową CO
	IF wPompaCO <> wPompaCOZaraportowana THEN
		wPompaCOZaraportowana := wPompaCO;
		fnKomunikatDaneDodaj_xOverFlow(sDane := sDane , sAtrybut := 'POMPA=' , sWartosc := WORD_TO_STRING(wPompaCO) , xOverFlow := xOverFlow);	
		IF xOverFlow = TRUE THEN
			fnZapiszKomunikat(	sCalyKomunikat := '' ,
						sTypKomunikatu := 'M' ,
						sMnemonik := sMnemonik ,
						sMACAdres := sMACAdres ,
						sIDNadawcy := sIdInstancji ,
						sIDOdbiorcy := sIdAplikacji ,
						sDaneZapasowe := sDaneZapasowe ,
						sDane := sDane ,
						arTablicaKomunikatow := arTablicaKomunikatow ,
						intTablicaKomunikatowZnacznikZapisu := intTablicaKomunikatowZnacznikZapisu ,
						intTablicaKomunikatowRozmiar := intTablicaKomunikatowRozmiar ,
						sWyslanyKomunikat := sWyslanyKomunikatDummy);
			sDane := '';
		END_IF	
	END_IF
	// Stan wyjść sterujących siłownikiem zaworu mieszającego CO
	IF wZaworCOZamkniecie <> wZaworCOZamkniecieZaraportowana THEN
		wZaworCOZamkniecieZaraportowana := wZaworCOZamkniecie;
		fnKomunikatDaneDodaj_xOverFlow(sDane := sDane , sAtrybut := 'ZAWORCOZAM=' , sWartosc := WORD_TO_STRING(wZaworCOZamkniecie) , xOverFlow := xOverFlow);	
		IF xOverFlow = TRUE THEN
			fnZapiszKomunikat(	sCalyKomunikat := '' ,
						sTypKomunikatu := 'M' ,
						sMnemonik := sMnemonik ,
						sMACAdres := sMACAdres ,
						sIDNadawcy := sIdInstancji ,
						sIDOdbiorcy := sIdAplikacji ,
						sDaneZapasowe := sDaneZapasowe ,
						sDane := sDane ,
						arTablicaKomunikatow := arTablicaKomunikatow ,
						intTablicaKomunikatowZnacznikZapisu := intTablicaKomunikatowZnacznikZapisu ,
						intTablicaKomunikatowRozmiar := intTablicaKomunikatowRozmiar ,
						sWyslanyKomunikat := sWyslanyKomunikatDummy);
			sDane := '';
		END_IF	
	END_IF
	// Stan wyjść sterujących siłownikiem zaworu mieszającego CO
	IF wZaworCOOtwarcie <> wZaworCOOtwarcieZaraportowana THEN
		wZaworCOOtwarcieZaraportowana := wZaworCOOtwarcie;
		fnKomunikatDaneDodaj_xOverFlow(sDane := sDane , sAtrybut := 'ZAWORCOOTW=' , sWartosc := WORD_TO_STRING(wZaworCOOtwarcie) , xOverFlow := xOverFlow);	
		IF xOverFlow = TRUE THEN
			fnZapiszKomunikat(	sCalyKomunikat := '' ,
						sTypKomunikatu := 'M' ,
						sMnemonik := sMnemonik ,
						sMACAdres := sMACAdres ,
						sIDNadawcy := sIdInstancji ,
						sIDOdbiorcy := sIdAplikacji ,
						sDaneZapasowe := sDaneZapasowe ,
						sDane := sDane ,
						arTablicaKomunikatow := arTablicaKomunikatow ,
						intTablicaKomunikatowZnacznikZapisu := intTablicaKomunikatowZnacznikZapisu ,
						intTablicaKomunikatowRozmiar := intTablicaKomunikatowRozmiar ,
						sWyslanyKomunikat := sWyslanyKomunikatDummy);
			sDane := '';
		END_IF	
	END_IF	
	IF xSezonGrzewczy <> xSezonGrzewczyZaraportowana THEN
		xSezonGrzewczyZaraportowana := xSezonGrzewczy;
		fnKomunikatDaneDodaj_xOverFlow(sDane := sDane , sAtrybut := 'SEZONGRZ=' , sWartosc := BOOL_TO_STRING(xSezonGrzewczy) , xOverFlow := xOverFlow);	
		IF xOverFlow = TRUE THEN
			fnZapiszKomunikat(	sCalyKomunikat := '' ,
						sTypKomunikatu := 'M' ,
						sMnemonik := sMnemonik ,
						sMACAdres := sMACAdres ,
						sIDNadawcy := sIdInstancji ,
						sIDOdbiorcy := sIdAplikacji ,
						sDaneZapasowe := sDaneZapasowe ,
						sDane := sDane ,
						arTablicaKomunikatow := arTablicaKomunikatow ,
						intTablicaKomunikatowZnacznikZapisu := intTablicaKomunikatowZnacznikZapisu ,
						intTablicaKomunikatowRozmiar := intTablicaKomunikatowRozmiar ,
						sWyslanyKomunikat := sWyslanyKomunikatDummy);
			sDane := '';
		END_IF	
	END_IF	
	IF rTemperaturaSrednia1Dzien <> rTemperaturaSrednia1DzienZaraportowana THEN
		rTemperaturaSrednia1DzienZaraportowana := rTemperaturaSrednia1Dzien;
		fnKomunikatDaneDodaj_xOverFlow(sDane := sDane , sAtrybut := 'TEMPSR1DZ=' , sWartosc := REAL_TO_STRING(rTemperaturaSrednia1Dzien + 273.15) , xOverFlow := xOverFlow);	
		IF xOverFlow = TRUE THEN
			fnZapiszKomunikat(	sCalyKomunikat := '' ,
						sTypKomunikatu := 'M' ,
						sMnemonik := sMnemonik ,
						sMACAdres := sMACAdres ,
						sIDNadawcy := sIdInstancji ,
						sIDOdbiorcy := sIdAplikacji ,
						sDaneZapasowe := sDaneZapasowe ,
						sDane := sDane ,
						arTablicaKomunikatow := arTablicaKomunikatow ,
						intTablicaKomunikatowZnacznikZapisu := intTablicaKomunikatowZnacznikZapisu ,
						intTablicaKomunikatowRozmiar := intTablicaKomunikatowRozmiar ,
						sWyslanyKomunikat := sWyslanyKomunikatDummy);
			sDane := '';
		END_IF	
	END_IF	
	IF sDane <> '' AND xPoInicjalizacji THEN
		fnZapiszKomunikat(	sCalyKomunikat := '' ,
							sTypKomunikatu := 'M' ,
							sMnemonik := sMnemonik ,
							sMACAdres := sMACAdres ,
							sIDNadawcy := sIdInstancji ,
							sIDOdbiorcy := sIdAplikacji ,
							sDaneZapasowe := sDaneZapasowe ,
							sDane := sDane ,
							arTablicaKomunikatow := arTablicaKomunikatow ,
							intTablicaKomunikatowZnacznikZapisu := intTablicaKomunikatowZnacznikZapisu ,
							intTablicaKomunikatowRozmiar := intTablicaKomunikatowRozmiar ,
							sWyslanyKomunikat := sWyslanyKomunikat);
	END_IF
END_IF
	
// Alarm braku komunikacji MODBUS 
IF arErrorStan[enumPPPSFriskoATTOM1SError.BrakKomunikacji] <> enumAlarmWartosc.StanAlarmowy AND arModbusStatusKomunikacji[bAdres] = enumModbusStatus.BrakKomunikacji THEN
	arErrorStan[enumPPPSFriskoATTOM1SError.BrakKomunikacji] := enumAlarmWartosc.StanAlarmowy;
	arErrorKlasa[enumPPPSFriskoATTOM1SError.BrakKomunikacji] := enumPPPSFriskoATTOM1SErrorKlasa.BrakKomunikacji;
	IF xPoInicjalizacji THEN
		fnZapiszKomunikat(	sCalyKomunikat := '' ,
							sTypKomunikatu := 'E' ,
							sMnemonik := sMnemonik ,
							sMACAdres := sMACAdres ,
							sIDNadawcy := sIdInstancji ,
							sIDOdbiorcy := sIdAplikacji ,
							sDaneZapasowe := sDaneZapasowe ,
							sDane := fnKomunikatDaneError(xAktywny := TRUE , intKlasa := enumPPPSFriskoATTOM1SErrorKlasa.BrakKomunikacji , intNumer := enumPPPSFriskoATTOM1SError.BrakKomunikacji),
							arTablicaKomunikatow := arTablicaKomunikatow ,
							intTablicaKomunikatowZnacznikZapisu := intTablicaKomunikatowZnacznikZapisu ,
							intTablicaKomunikatowRozmiar := intTablicaKomunikatowRozmiar ,
							sWyslanyKomunikat := sWyslanyKomunikatDummy);
	END_IF
END_IF
IF arErrorStan[enumPPPSFriskoATTOM1SError.BrakKomunikacji] <> enumAlarmWartosc.StanNormalny AND arModbusStatusKomunikacji[bAdres] = enumModbusStatus.KomunikacjaPrawidlowa THEN
	arErrorStan[enumPPPSFriskoATTOM1SError.BrakKomunikacji] := enumAlarmWartosc.StanNormalny;
	arErrorKlasa[enumPPPSFriskoATTOM1SError.BrakKomunikacji] := enumPPPSFriskoATTOM1SErrorKlasa.BrakKomunikacji;
	IF xPoInicjalizacji THEN
		fnZapiszKomunikat(	sCalyKomunikat := '' ,
							sTypKomunikatu := 'E' ,
							sMnemonik := sMnemonik ,
							sMACAdres := sMACAdres ,
							sIDNadawcy := sIdInstancji ,
							sIDOdbiorcy := sIdAplikacji ,
							sDaneZapasowe := sDaneZapasowe ,
							sDane := fnKomunikatDaneError(xAktywny := FALSE , intKlasa := enumPPPSFriskoATTOM1SErrorKlasa.BrakKomunikacji , intNumer := enumPPPSFriskoATTOM1SError.BrakKomunikacji),
							arTablicaKomunikatow := arTablicaKomunikatow ,
							intTablicaKomunikatowZnacznikZapisu := intTablicaKomunikatowZnacznikZapisu ,
							intTablicaKomunikatowRozmiar := intTablicaKomunikatowRozmiar ,
							sWyslanyKomunikat := sWyslanyKomunikatDummy);
	END_IF
END_IF
	
// Alarm czujnika temperatury zewnętrznej 
IF arErrorStan[enumPPPSFriskoATTOM1SError.AlarmCzujnikaZewnetrznego] <> enumAlarmWartosc.StanAlarmowy AND xBladBrakZmianyTemperaturyZewnetrznej THEN
	arErrorStan[enumPPPSFriskoATTOM1SError.AlarmCzujnikaZewnetrznego] := enumAlarmWartosc.StanAlarmowy;
	arErrorKlasa[enumPPPSFriskoATTOM1SError.AlarmCzujnikaZewnetrznego] := enumPPPSFriskoATTOM1SErrorKlasa.AlarmCzujnikaZewnetrznego;
	IF xPoInicjalizacji THEN
		fnZapiszKomunikat(	sCalyKomunikat := '' ,
							sTypKomunikatu := 'E' ,
							sMnemonik := sMnemonik ,
							sMACAdres := sMACAdres ,
							sIDNadawcy := sIdInstancji ,
							sIDOdbiorcy := sIdAplikacji ,
							sDaneZapasowe := sDaneZapasowe ,
							sDane := fnKomunikatDaneError(xAktywny := TRUE , intKlasa := enumPPPSFriskoATTOM1SErrorKlasa.AlarmCzujnikaZewnetrznego , intNumer := enumPPPSFriskoATTOM1SError.AlarmCzujnikaZewnetrznego),
							arTablicaKomunikatow := arTablicaKomunikatow ,
							intTablicaKomunikatowZnacznikZapisu := intTablicaKomunikatowZnacznikZapisu ,
							intTablicaKomunikatowRozmiar := intTablicaKomunikatowRozmiar ,
							sWyslanyKomunikat := sWyslanyKomunikatDummy);
	END_IF
END_IF
IF arErrorStan[enumPPPSFriskoATTOM1SError.AlarmCzujnikaZewnetrznego] <> enumAlarmWartosc.StanNormalny AND NOT xBladBrakZmianyTemperaturyZewnetrznej THEN
	arErrorStan[enumPPPSFriskoATTOM1SError.AlarmCzujnikaZewnetrznego] := enumAlarmWartosc.StanNormalny;
	arErrorKlasa[enumPPPSFriskoATTOM1SError.AlarmCzujnikaZewnetrznego] := enumPPPSFriskoATTOM1SErrorKlasa.AlarmCzujnikaZewnetrznego;
	IF xPoInicjalizacji THEN
		fnZapiszKomunikat(	sCalyKomunikat := '' ,
							sTypKomunikatu := 'E' ,
							sMnemonik := sMnemonik ,
							sMACAdres := sMACAdres ,
							sIDNadawcy := sIdInstancji ,
							sIDOdbiorcy := sIdAplikacji ,
							sDaneZapasowe := sDaneZapasowe ,
							sDane := fnKomunikatDaneError(xAktywny := FALSE , intKlasa := enumPPPSFriskoATTOM1SErrorKlasa.AlarmCzujnikaZewnetrznego , intNumer := enumPPPSFriskoATTOM1SError.AlarmCzujnikaZewnetrznego),
							arTablicaKomunikatow := arTablicaKomunikatow ,
							intTablicaKomunikatowZnacznikZapisu := intTablicaKomunikatowZnacznikZapisu ,
							intTablicaKomunikatowRozmiar := intTablicaKomunikatowRozmiar ,
							sWyslanyKomunikat := sWyslanyKomunikatDummy);
	END_IF
END_IF
	
// Alarm czujnika temperatury zasilania
IF arErrorStan[enumPPPSFriskoATTOM1SError.AlarmCzujnikaZasilaniaObwoduCO] <> enumAlarmWartosc.StanAlarmowy AND xBladBrakZmianyTemperaturyZasilaniaObieguCO THEN
	arErrorStan[enumPPPSFriskoATTOM1SError.AlarmCzujnikaZasilaniaObwoduCO] := enumAlarmWartosc.StanAlarmowy;
	arErrorKlasa[enumPPPSFriskoATTOM1SError.AlarmCzujnikaZasilaniaObwoduCO] := enumPPPSFriskoATTOM1SErrorKlasa.AlarmCzujnikaZasilaniaObwoduCO;
	IF xPoInicjalizacji THEN
		fnZapiszKomunikat(	sCalyKomunikat := '' ,
							sTypKomunikatu := 'E' ,
							sMnemonik := sMnemonik ,
							sMACAdres := sMACAdres ,
							sIDNadawcy := sIdInstancji ,
							sIDOdbiorcy := sIdAplikacji ,
							sDaneZapasowe := sDaneZapasowe ,
							sDane := fnKomunikatDaneError(xAktywny := TRUE , intKlasa := enumPPPSFriskoATTOM1SErrorKlasa.AlarmCzujnikaZasilaniaObwoduCO , intNumer := enumPPPSFriskoATTOM1SError.AlarmCzujnikaZasilaniaObwoduCO),
							arTablicaKomunikatow := arTablicaKomunikatow ,
							intTablicaKomunikatowZnacznikZapisu := intTablicaKomunikatowZnacznikZapisu ,
							intTablicaKomunikatowRozmiar := intTablicaKomunikatowRozmiar ,
							sWyslanyKomunikat := sWyslanyKomunikatDummy);
	END_IF
END_IF
IF arErrorStan[enumPPPSFriskoATTOM1SError.AlarmCzujnikaZasilaniaObwoduCO] <> enumAlarmWartosc.StanNormalny AND NOT xBladBrakZmianyTemperaturyZasilaniaObieguCO THEN
	arErrorStan[enumPPPSFriskoATTOM1SError.AlarmCzujnikaZasilaniaObwoduCO] := enumAlarmWartosc.StanNormalny;
	arErrorKlasa[enumPPPSFriskoATTOM1SError.AlarmCzujnikaZasilaniaObwoduCO] := enumPPPSFriskoATTOM1SErrorKlasa.AlarmCzujnikaZasilaniaObwoduCO;
	IF xPoInicjalizacji THEN
		fnZapiszKomunikat(	sCalyKomunikat := '' ,
							sTypKomunikatu := 'E' ,
							sMnemonik := sMnemonik ,
							sMACAdres := sMACAdres ,
							sIDNadawcy := sIdInstancji ,
							sIDOdbiorcy := sIdAplikacji ,
							sDaneZapasowe := sDaneZapasowe ,
							sDane := fnKomunikatDaneError(xAktywny := FALSE , intKlasa := enumPPPSFriskoATTOM1SErrorKlasa.AlarmCzujnikaZasilaniaObwoduCO , intNumer := enumPPPSFriskoATTOM1SError.AlarmCzujnikaZasilaniaObwoduCO),
							arTablicaKomunikatow := arTablicaKomunikatow ,
							intTablicaKomunikatowZnacznikZapisu := intTablicaKomunikatowZnacznikZapisu ,
							intTablicaKomunikatowRozmiar := intTablicaKomunikatowRozmiar ,
							sWyslanyKomunikat := sWyslanyKomunikatDummy);
	END_IF
END_IF
	
// Alarm braku osiągnięcia temperatury zadanej
IF arErrorStan[enumPPPSFriskoATTOM1SError.BrakOsiagnieciaTemperaturyCO] <> enumAlarmWartosc.StanAlarmowy AND xBladBrakOsiagnieciaTemperauryZadanejCO THEN
	arErrorStan[enumPPPSFriskoATTOM1SError.BrakOsiagnieciaTemperaturyCO] := enumAlarmWartosc.StanAlarmowy;
	arErrorKlasa[enumPPPSFriskoATTOM1SError.BrakOsiagnieciaTemperaturyCO] := enumPPPSFriskoATTOM1SErrorKlasa.BrakOsiagnieciaTemperaturyCO;
	IF xPoInicjalizacji THEN
		fnZapiszKomunikat(	sCalyKomunikat := '' ,
							sTypKomunikatu := 'E' ,
							sMnemonik := sMnemonik ,
							sMACAdres := sMACAdres ,
							sIDNadawcy := sIdInstancji ,
							sIDOdbiorcy := sIdAplikacji ,
							sDaneZapasowe := sDaneZapasowe ,
							sDane := fnKomunikatDaneError(xAktywny := TRUE , intKlasa := enumPPPSFriskoATTOM1SErrorKlasa.BrakOsiagnieciaTemperaturyCO , intNumer := enumPPPSFriskoATTOM1SError.BrakOsiagnieciaTemperaturyCO),
							arTablicaKomunikatow := arTablicaKomunikatow ,
							intTablicaKomunikatowZnacznikZapisu := intTablicaKomunikatowZnacznikZapisu ,
							intTablicaKomunikatowRozmiar := intTablicaKomunikatowRozmiar ,
							sWyslanyKomunikat := sWyslanyKomunikatDummy);
	END_IF
END_IF
IF arErrorStan[enumPPPSFriskoATTOM1SError.BrakOsiagnieciaTemperaturyCO] <> enumAlarmWartosc.StanNormalny AND NOT xBladBrakOsiagnieciaTemperauryZadanejCO THEN
	arErrorStan[enumPPPSFriskoATTOM1SError.BrakOsiagnieciaTemperaturyCO] := enumAlarmWartosc.StanNormalny;
	arErrorKlasa[enumPPPSFriskoATTOM1SError.BrakOsiagnieciaTemperaturyCO] := enumPPPSFriskoATTOM1SErrorKlasa.BrakOsiagnieciaTemperaturyCO;
	IF xPoInicjalizacji THEN
		fnZapiszKomunikat(	sCalyKomunikat := '' ,
							sTypKomunikatu := 'E' ,
							sMnemonik := sMnemonik ,
							sMACAdres := sMACAdres ,
							sIDNadawcy := sIdInstancji ,
							sIDOdbiorcy := sIdAplikacji ,
							sDaneZapasowe := sDaneZapasowe ,
							sDane := fnKomunikatDaneError(xAktywny := FALSE , intKlasa := enumPPPSFriskoATTOM1SErrorKlasa.BrakOsiagnieciaTemperaturyCO , intNumer := enumPPPSFriskoATTOM1SError.BrakOsiagnieciaTemperaturyCO),
							arTablicaKomunikatow := arTablicaKomunikatow ,
							intTablicaKomunikatowZnacznikZapisu := intTablicaKomunikatowZnacznikZapisu ,
							intTablicaKomunikatowRozmiar := intTablicaKomunikatowRozmiar ,
							sWyslanyKomunikat := sWyslanyKomunikatDummy);
	END_IF
END_IF

// Alarm braku wymaganej ilości pomiarów do obliczenia średniej temperatury
IF arErrorStan[enumPPPSFriskoATTOM1SError.BladIloscPomiarowTemperatury] <> enumAlarmWartosc.StanAlarmowy AND xBladIloscPomiarowTemperatury THEN
	arErrorStan[enumPPPSFriskoATTOM1SError.BladIloscPomiarowTemperatury] := enumAlarmWartosc.StanAlarmowy;
	arErrorKlasa[enumPPPSFriskoATTOM1SError.BladIloscPomiarowTemperatury] := enumPPPSFriskoATTOM1SErrorKlasa.BladIloscPomiarowTemperatury;
	IF xPoInicjalizacji THEN
		fnZapiszKomunikat(	sCalyKomunikat := '' ,
							sTypKomunikatu := 'E' ,
							sMnemonik := sMnemonik ,
							sMACAdres := sMACAdres ,
							sIDNadawcy := sIdInstancji ,
							sIDOdbiorcy := sIdAplikacji ,
							sDaneZapasowe := sDaneZapasowe ,
							sDane := fnKomunikatDaneError(xAktywny := TRUE , intKlasa := enumPPPSFriskoATTOM1SErrorKlasa.BladIloscPomiarowTemperatury , intNumer := enumPPPSFriskoATTOM1SError.BladIloscPomiarowTemperatury),
							arTablicaKomunikatow := arTablicaKomunikatow ,
							intTablicaKomunikatowZnacznikZapisu := intTablicaKomunikatowZnacznikZapisu ,
							intTablicaKomunikatowRozmiar := intTablicaKomunikatowRozmiar ,
							sWyslanyKomunikat := sWyslanyKomunikatDummy);
	END_IF
END_IF
          
END_FUNCTION_BLOCK
